LIN {X 0,Y 305.687,Z 241.405,A -85,B 0,C 180,E1 -15834.723,E2 -15834.723} C_VEL
LIN {X 0,Y 305.955,Z 241.369,A -85,B 0,C 180,E1 -15838.684,E2 -15838.684} C_VEL
LIN {X 0,Y 305.953,Z 241.364,A -85,B 0,C 180,E1 -15841.316,E2 -15841.316} C_VEL
LIN {X 0,Y 305.687,Z 241.402,A -85,B 0,C 180,E1 -15845.276,E2 -15845.276} C_VEL
LIN {X 0,Y 305.811,Z 241.392,A -85,B 0,C 180,E1 -15847.926,E2 -15847.926} C_VEL
LIN {X 0,Y 305.601,Z 241.415,A -85,B 0,C 180,E1 -15851.945,E2 -15851.945} C_VEL
LIN {X 0,Y 305.635,Z 241.408,A -85,B 0,C 180,E1 -15855.035,E2 -15855.035} C_VEL
LIN {X 0,Y 305.575,Z 241.418,A -85,B 0,C 180,E1 -15859.445,E2 -15859.445} C_VEL
LIN {X 0,Y 305.489,Z 241.428,A -85,B 0,C 180,E1 -15863.042,E2 -15863.042} C_VEL
LIN {X 0,Y 305.545,Z 241.427,A -85,B 0,C 180,E1 -15866.227,E2 -15866.227} C_VEL
LIN {X 0,Y 305.493,Z 241.428,A -85,B 0,C 180,E1 -15869.05,E2 -15869.05} C_VEL
LIN {X 0,Y 305.442,Z 241.437,A -85,B 0,C 180,E1 -15871.952,E2 -15871.952} C_VEL
LIN {X 0,Y 305.46,Z 241.433,A -85,B 0,C 180,E1 -15875.114,E2 -15875.114} C_VEL
LIN {X 0,Y 305.448,Z 241.439,A -85,B 0,C 180,E1 -15878.529,E2 -15878.529} C_VEL
LIN {X 0,Y 305.453,Z 241.434,A -85,B 0,C 180,E1 -15882.586,E2 -15882.586} C_VEL
LIN {X 0,Y 305.472,Z 241.432,A -85,B 0,C 180,E1 -15887.411,E2 -15887.411} C_VEL
LIN {X 0,Y 305.495,Z 241.428,A -85,B 0,C 180,E1 -15891.601,E2 -15891.601} C_VEL
LIN {X 0,Y 305.462,Z 241.439,A -85,B 0,C 180,E1 -15894.887,E2 -15894.887} C_VEL
LIN {X 0,Y 305.506,Z 241.55,A -85,B 0,C 180,E1 -15897.52,E2 -15897.52} C_VEL
LIN {X 0,Y 307.816,Z 252.02,A -85,B 0,C 180,E1 -15900.845,E2 -15900.845} C_VEL
LIN {X 0,Y 309.592,Z 261.539,A -85,B 0,C 180,E1 -15903.726,E2 -15903.726} C_VEL
LIN {X 0,Y 309.871,Z 264.214,A -85,B 0,C 180,E1 -15904.504,E2 -15904.504} C_VEL
LIN {X 0,Y 315.45,Z 298.867,A -85,B 0,C 180,E1 -15905.809,E2 -15905.809} C_VEL
LIN {X 0,Y 316.306,Z 306.855,A -85,B 0,C 180,E1 -15906.07,E2 -15906.07} C_VEL
LIN {X 0,Y 314.598,Z 373.309,A -85,B 0,C 180,E1 -15907.645,E2 -15907.645} C_VEL
LIN {X 0,Y 313.755,Z 386.795,A -85,B 0,C 180,E1 -15908.223,E2 -15908.223} C_VEL
LIN {X 0,Y 312.61,Z 399.148,A -85,B 0,C 180,E1 -15909.004,E2 -15909.004} C_VEL
LIN {X 0,Y 311.362,Z 411.031,A -85,B 0,C 180,E1 -15910.038,E2 -15910.038} C_VEL
LIN {X 0,Y 309.959,Z 422.47,A -85,B 0,C 180,E1 -15911.321,E2 -15911.321} C_VEL
LIN {X 0,Y 308.58,Z 432.784,A -85,B 0,C 180,E1 -15912.778,E2 -15912.778} C_VEL
LIN {X 0,Y 307.385,Z 442.048,A -85,B 0,C 180,E1 -15914.416,E2 -15914.416} C_VEL
LIN {X 0,Y 306.04,Z 451.048,A -85,B 0,C 180,E1 -15916.386,E2 -15916.386} C_VEL
LIN {X 0,Y 304.97,Z 458.282,A -85,B 0,C 180,E1 -15918.367,E2 -15918.367} C_VEL
LIN {X 0,Y 304.41,Z 463.162,A -85,B 0,C 180,E1 -15920.029,E2 -15920.029} C_VEL
LIN {X 0,Y 303.949,Z 467.893,A -85,B 0,C 180,E1 -15922.026,E2 -15922.026} C_VEL
LIN {X 0,Y 303.625,Z 472.136,A -85,B 0,C 180,E1 -15924.456,E2 -15924.456} C_VEL
LIN {X 0,Y 303.63,Z 474.065,A -85,B 0,C 180,E1 -15926.018,E2 -15926.018} C_VEL
LIN {X 0,Y 303.607,Z 475.267,A -85,B 0,C 180,E1 -15927.347,E2 -15927.347} C_VEL
LIN {X 0,Y 303.574,Z 476.018,A -85,B 0,C 180,E1 -15928.674,E2 -15928.674} C_VEL
LIN {X 0,Y 303.603,Z 476.368,A -85,B 0,C 180,E1 -15930,E2 -15930} C_VEL
LIN {X 0,Y 303.602,Z 475.896,A -85,B 0,C 180,E1 -15932.654,E2 -15932.654} C_VEL
LIN {X 0,Y 303.592,Z 475.028,A -85,B 0,C 180,E1 -15933.982,E2 -15933.982} C_VEL
LIN {X 0,Y 303.739,Z 472.071,A -85,B 0,C 180,E1 -15936.644,E2 -15936.644} C_VEL
LIN {X 0,Y 304.142,Z 468.709,A -85,B 0,C 180,E1 -15938.639,E2 -15938.639} C_VEL
LIN {X 0,Y 304.728,Z 464.278,A -85,B 0,C 180,E1 -15940.632,E2 -15940.632} C_VEL
LIN {X 0,Y 305.609,Z 458.66,A -85,B 0,C 180,E1 -15942.619,E2 -15942.619} C_VEL
LIN {X 0,Y 306.952,Z 451.662,A -85,B 0,C 180,E1 -15944.588,E2 -15944.588} C_VEL
LIN {X 0,Y 308.292,Z 443.612,A -85,B 0,C 180,E1 -15946.41,E2 -15946.41} C_VEL
LIN {X 0,Y 309.891,Z 433.972,A -85,B 0,C 180,E1 -15948.17,E2 -15948.17} C_VEL
LIN {X 0,Y 311.519,Z 424.167,A -85,B 0,C 180,E1 -15949.608,E2 -15949.608} C_VEL
LIN {X 0,Y 313.136,Z 413.41,A -85,B 0,C 180,E1 -15950.873,E2 -15950.873} C_VEL
LIN {X 0,Y 314.748,Z 401.372,A -85,B 0,C 180,E1 -15951.963,E2 -15951.963} C_VEL
LIN {X 0,Y 316.079,Z 388.872,A -85,B 0,C 180,E1 -15952.813,E2 -15952.813} C_VEL
LIN {X 0,Y 317.128,Z 375.767,A -85,B 0,C 180,E1 -15953.423,E2 -15953.423} C_VEL
LIN {X 0,Y 317.823,Z 359.088,A -85,B 0,C 180,E1 -15953.878,E2 -15953.878} C_VEL
LIN {X 0,Y 319.113,Z 304.9,A -85,B 0,C 180,E1 -15955.164,E2 -15955.164} C_VEL
LIN {X 0,Y 315.677,Z 283.465,A -85,B 0,C 180,E1 -15956.063,E2 -15956.063} C_VEL
LIN {X 0,Y 312.582,Z 268.833,A -85,B 0,C 180,E1 -15956.769,E2 -15956.769} C_VEL
LIN {X 0,Y 310.331,Z 263.131,A -85,B 0,C 180,E1 -15957.165,E2 -15957.165} C_VEL
LIN {X 0,Y 308.466,Z 253.823,A -85,B 0,C 180,E1 -15960.082,E2 -15960.082} C_VEL
LIN {X 0,Y 306.055,Z 243.759,A -85,B 0,C 180,E1 -15963.444,E2 -15963.444} C_VEL
LIN {X 0,Y 305.478,Z 241.436,A -85,B 0,C 180,E1 -15964.32,E2 -15964.32} C_VEL
LIN {X 0,Y 305.476,Z 241.432,A -85,B 0,C 180,E1 -15968.402,E2 -15968.402} C_VEL
LIN {X 0,Y 305.455,Z 241.433,A -85,B 0,C 180,E1 -15972.586,E2 -15972.586} C_VEL
LIN {X 0,Y 305.426,Z 241.441,A -85,B 0,C 180,E1 -15976.345,E2 -15976.345} C_VEL
LIN {X 0,Y 305.458,Z 241.436,A -85,B 0,C 180,E1 -15979.892,E2 -15979.892} C_VEL
LIN {X 0,Y 305.481,Z 241.431,A -85,B 0,C 180,E1 -15983.631,E2 -15983.631} C_VEL
LIN {X 0,Y 305.465,Z 241.433,A -85,B 0,C 180,E1 -15986.483,E2 -15986.483} C_VEL
LIN {X 0,Y 305.458,Z 241.432,A -85,B 0,C 180,E1 -15989.59,E2 -15989.59} C_VEL
LIN {X 0,Y 305.518,Z 241.42,A -85,B 0,C 180,E1 -15992.608,E2 -15992.608} C_VEL
LIN {X 0,Y 305.508,Z 241.427,A -85,B 0,C 180,E1 -15995.539,E2 -15995.539} C_VEL
LIN {X 0,Y 305.519,Z 241.426,A -85,B 0,C 180,E1 -15999.815,E2 -15999.815} C_VEL
LIN {X 0,Y 305.574,Z 241.416,A -85,B 0,C 180,E1 -16002.603,E2 -16002.603} C_VEL
LIN {X 0,Y 305.649,Z 241.401,A -85,B 0,C 180,E1 -16005.349,E2 -16005.349} C_VEL
LIN {X 0,Y 305.638,Z 241.407,A -85,B 0,C 180,E1 -16009.4,E2 -16009.4} C_VEL
LIN {X 0,Y 305.808,Z 241.389,A -85,B 0,C 180,E1 -16012.074,E2 -16012.074} C_VEL
LIN {X 0,Y 305.686,Z 241.399,A -85,B 0,C 180,E1 -16014.724,E2 -16014.724} C_VEL
LIN {X 0,Y 305.955,Z 241.369,A -85,B 0,C 180,E1 -16018.684,E2 -16018.684} C_VEL
LIN {X 0,Y 305.957,Z 241.374,A -85,B 0,C 180,E1 -16021.316,E2 -16021.316} C_VEL
LIN {X 0,Y 305.851,Z 241.387,A -85,B 0,C 180,E1 -16026.598,E2 -16026.598} C_VEL
LIN {X 0,Y 305.736,Z 241.401,A -85,B 0,C 180,E1 -16029.26,E2 -16029.26} C_VEL
LIN {X 0,Y 305.589,Z 241.42,A -85,B 0,C 180,E1 -16033.296,E2 -16033.296} C_VEL
LIN {X 0,Y 305.594,Z 241.415,A -85,B 0,C 180,E1 -16036.02,E2 -16036.02} C_VEL
LIN {X 0,Y 305.576,Z 241.421,A -85,B 0,C 180,E1 -16039.444,E2 -16039.444} C_VEL
LIN {X 0,Y 305.486,Z 241.432,A -85,B 0,C 180,E1 -16043.04,E2 -16043.04} C_VEL
LIN {X 0,Y 305.478,Z 241.432,A -85,B 0,C 180,E1 -16046.201,E2 -16046.201} C_VEL
LIN {X 0,Y 305.463,Z 241.425,A -85,B 0,C 180,E1 -16049.039,E2 -16049.039} C_VEL
LIN {X 0,Y 305.437,Z 241.433,A -85,B 0,C 180,E1 -16051.953,E2 -16051.953} C_VEL
LIN {X 0,Y 305.509,Z 241.449,A -85,B 0,C 180,E1 -16054.963,E2 -16054.963} C_VEL
LIN {X 0,Y 307.325,Z 248.984,A -85,B 0,C 180,E1 -16057.56,E2 -16057.56} C_VEL
LIN {X 0,Y 314.914,Z 265.656,A -85,B 0,C 180,E1 -16058.826,E2 -16058.826} C_VEL
LIN {X 0,Y 318.632,Z 275.459,A -85,B 0,C 180,E1 -16059.458,E2 -16059.458} C_VEL
LIN {X 0,Y 319.852,Z 282.666,A -85,B 0,C 180,E1 -16059.766,E2 -16059.766} C_VEL
LIN {X 0,Y 317.555,Z 356.862,A -85,B 0,C 180,E1 -16061.521,E2 -16061.521} C_VEL
LIN {X 0,Y 316.73,Z 370.282,A -85,B 0,C 180,E1 -16062.098,E2 -16062.098} C_VEL
LIN {X 0,Y 315.633,Z 382.988,A -85,B 0,C 180,E1 -16062.909,E2 -16062.909} C_VEL
LIN {X 0,Y 314.192,Z 395.492,A -85,B 0,C 180,E1 -16064.007,E2 -16064.007} C_VEL
LIN {X 0,Y 312.768,Z 405.819,A -85,B 0,C 180,E1 -16065.17,E2 -16065.17} C_VEL
LIN {X 0,Y 311.245,Z 415.778,A -85,B 0,C 180,E1 -16066.566,E2 -16066.566} C_VEL
LIN {X 0,Y 309.825,Z 423.975,A -85,B 0,C 180,E1 -16067.969,E2 -16067.969} C_VEL
LIN {X 0,Y 308.179,Z 433.065,A -85,B 0,C 180,E1 -16069.891,E2 -16069.891} C_VEL
LIN {X 0,Y 306.879,Z 440.278,A -85,B 0,C 180,E1 -16071.805,E2 -16071.805} C_VEL
LIN {X 0,Y 305.889,Z 445.559,A -85,B 0,C 180,E1 -16073.528,E2 -16073.528} C_VEL
LIN {X 0,Y 304.994,Z 450.479,A -85,B 0,C 180,E1 -16075.539,E2 -16075.539} C_VEL
LIN {X 0,Y 304.303,Z 454.817,A -85,B 0,C 180,E1 -16077.914,E2 -16077.914} C_VEL
LIN {X 0,Y 303.94,Z 456.818,A -85,B 0,C 180,E1 -16079.422,E2 -16079.422} C_VEL
LIN {X 0,Y 303.555,Z 458.759,A -85,B 0,C 180,E1 -16081.618,E2 -16081.618} C_VEL
LIN {X 0,Y 303.342,Z 459.607,A -85,B 0,C 180,E1 -16083.883,E2 -16083.883} C_VEL
LIN {X 0,Y 303.31,Z 459.554,A -85,B 0,C 180,E1 -16085.35,E2 -16085.35} C_VEL
LIN {X 0,Y 303.408,Z 458.277,A -85,B 0,C 180,E1 -16087.903,E2 -16087.903} C_VEL
LIN {X 0,Y 303.822,Z 455.551,A -85,B 0,C 180,E1 -16090.402,E2 -16090.402} C_VEL
LIN {X 0,Y 304.263,Z 452.031,A -85,B 0,C 180,E1 -16092.526,E2 -16092.526} C_VEL
LIN {X 0,Y 304.826,Z 447.343,A -85,B 0,C 180,E1 -16094.625,E2 -16094.625} C_VEL
LIN {X 0,Y 305.708,Z 441.312,A -85,B 0,C 180,E1 -16096.709,E2 -16096.709} C_VEL
LIN {X 0,Y 306.77,Z 433.714,A -85,B 0,C 180,E1 -16098.771,E2 -16098.771} C_VEL
LIN {X 0,Y 307.949,Z 425.894,A -85,B 0,C 180,E1 -16100.482,E2 -16100.482} C_VEL
LIN {X 0,Y 309.248,Z 416.482,A -85,B 0,C 180,E1 -16102.163,E2 -16102.163} C_VEL
LIN {X 0,Y 310.677,Z 405.452,A -85,B 0,C 180,E1 -16103.726,E2 -16103.726} C_VEL
LIN {X 0,Y 312.054,Z 394.084,A -85,B 0,C 180,E1 -16104.993,E2 -16104.993} C_VEL
LIN {X 0,Y 313.249,Z 381.694,A -85,B 0,C 180,E1 -16106.06,E2 -16106.06} C_VEL
LIN {X 0,Y 314.143,Z 368.704,A -85,B 0,C 180,E1 -16106.874,E2 -16106.874} C_VEL
LIN {X 0,Y 314.773,Z 356.239,A -85,B 0,C 180,E1 -16107.4,E2 -16107.4} C_VEL
LIN {X 0,Y 316.733,Z 280.316,A -85,B 0,C 180,E1 -16109.187,E2 -16109.187} C_VEL
LIN {X 0,Y 314.043,Z 267.159,A -85,B 0,C 180,E1 -16109.718,E2 -16109.718} C_VEL
LIN {X 0,Y 307.327,Z 248.529,A -85,B 0,C 180,E1 -16110.737,E2 -16110.737} C_VEL
LIN {X 0,Y 305.729,Z 241.405,A -85,B 0,C 180,E1 -16113.212,E2 -16113.212} C_VEL
LIN {X 0,Y 305.789,Z 241.395,A -85,B 0,C 180,E1 -16116.599,E2 -16116.599} C_VEL
LIN {X 0,Y 305.696,Z 241.406,A -85,B 0,C 180,E1 -16119.261,E2 -16119.261} C_VEL
LIN {X 0,Y 305.591,Z 241.419,A -85,B 0,C 180,E1 -16123.296,E2 -16123.296} C_VEL
LIN {X 0,Y 305.596,Z 241.421,A -85,B 0,C 180,E1 -16126.02,E2 -16126.02} C_VEL
LIN {X 0,Y 305.577,Z 241.422,A -85,B 0,C 180,E1 -16129.444,E2 -16129.444} C_VEL
LIN {X 0,Y 305.487,Z 241.427,A -85,B 0,C 180,E1 -16133.039,E2 -16133.039} C_VEL
LIN {X 0,Y 305.476,Z 241.433,A -85,B 0,C 180,E1 -16136.199,E2 -16136.199} C_VEL
LIN {X 0,Y 305.459,Z 241.43,A -85,B 0,C 180,E1 -16139.037,E2 -16139.037} C_VEL
LIN {X 0,Y 305.437,Z 241.441,A -85,B 0,C 180,E1 -16141.952,E2 -16141.952} C_VEL
LIN {X 0,Y 305.462,Z 241.43,A -85,B 0,C 180,E1 -16145.113,E2 -16145.113} C_VEL
LIN {X 0,Y 305.466,Z 241.433,A -85,B 0,C 180,E1 -16148.532,E2 -16148.532} C_VEL
LIN {X 0,Y 305.454,Z 241.431,A -85,B 0,C 180,E1 -16152.585,E2 -16152.585} C_VEL
LIN {X 0,Y 305.425,Z 241.438,A -85,B 0,C 180,E1 -16156.344,E2 -16156.344} C_VEL
LIN {X 0,Y 305.457,Z 241.438,A -85,B 0,C 180,E1 -16159.892,E2 -16159.892} C_VEL
LIN {X 0,Y 305.458,Z 241.432,A -85,B 0,C 180,E1 -16161.37,E2 -16161.37} C_VEL
LIN {X 0,Y 304.851,Z 241.512,A -85,B 0,C 180,E1 -16162.47,E2 -16162.47} C_VEL
LIN {X 0,Y 302.014,Z 241.864,A -85,B 0,C 180,E1 -16164.26,E2 -16164.26} C_VEL
LIN {X 0,Y 299.559,Z 242.166,A -85,B 0,C 180,E1 -16165.713,E2 -16165.713} C_VEL
LIN {X 0,Y 298.488,Z 242.299,A -85,B 0,C 180,E1 -16166.838,E2 -16166.838} C_VEL
LIN {X 0,Y 298.393,Z 242.311,A -85,B 0,C 180,E1 -16167.22,E2 -16167.22} C_VEL
LIN {X 0,Y 298.457,Z 242.309,A -85,B 0,C 180,E1 -16171.903,E2 -16171.903} C_VEL
LIN {X 0,Y 298.484,Z 242.294,A -85,B 0,C 180,E1 -16174.924,E2 -16174.924} C_VEL
LIN {X 0,Y 298.448,Z 242.303,A -85,B 0,C 180,E1 -16179.315,E2 -16179.315} C_VEL
LIN {X 0,Y 298.536,Z 242.3,A -85,B 0,C 180,E1 -16182.179,E2 -16182.179} C_VEL
LIN {X 0,Y 298.591,Z 242.286,A -85,B 0,C 180,E1 -16184.994,E2 -16184.994} C_VEL
LIN {X 0,Y 298.591,Z 242.277,A -85,B 0,C 180,E1 -16189.146,E2 -16189.146} C_VEL
LIN {X 0,Y 298.756,Z 242.266,A -85,B 0,C 180,E1 -16191.886,E2 -16191.886} C_VEL
LIN {X 0,Y 298.658,Z 242.282,A -85,B 0,C 180,E1 -16194.599,E2 -16194.599} C_VEL
LIN {X 0,Y 298.921,Z 242.245,A -85,B 0,C 180,E1 -16198.653,E2 -16198.653} C_VEL
LIN {X 0,Y 298.92,Z 242.239,A -85,B 0,C 180,E1 -16201.347,E2 -16201.347} C_VEL
LIN {X 0,Y 298.796,Z 242.264,A -85,B 0,C 180,E1 -16206.754,E2 -16206.754} C_VEL
LIN {X 0,Y 298.678,Z 242.277,A -85,B 0,C 180,E1 -16209.48,E2 -16209.48} C_VEL
LIN {X 0,Y 298.549,Z 242.286,A -85,B 0,C 180,E1 -16213.615,E2 -16213.615} C_VEL
LIN {X 0,Y 298.546,Z 242.297,A -85,B 0,C 180,E1 -16216.409,E2 -16216.409} C_VEL
LIN {X 0,Y 298.51,Z 242.299,A -85,B 0,C 180,E1 -16219.655,E2 -16219.655} C_VEL
LIN {X 0,Y 298.456,Z 242.304,A -85,B 0,C 180,E1 -16223.598,E2 -16223.598} C_VEL
LIN {X 0,Y 298.487,Z 242.303,A -85,B 0,C 180,E1 -16226.575,E2 -16226.575} C_VEL
LIN {X 0,Y 298.419,Z 242.309,A -85,B 0,C 180,E1 -16229.641,E2 -16229.641} C_VEL
LIN {X 0,Y 298.394,Z 242.313,A -85,B 0,C 180,E1 -16232.8,E2 -16232.8} C_VEL
LIN {X 0,Y 298.444,Z 242.308,A -85,B 0,C 180,E1 -16236.808,E2 -16236.808} C_VEL
LIN {X 0,Y 298.385,Z 242.313,A -85,B 0,C 180,E1 -16241.088,E2 -16241.088} C_VEL
LIN {X 0,Y 298.397,Z 242.311,A -85,B 0,C 180,E1 -16243.104,E2 -16243.104} C_VEL
LIN {X 0,Y 298.402,Z 242.314,A -85,B 0,C 180,E1 -16246.921,E2 -16246.921} C_VEL
LIN {X 0,Y 298.414,Z 242.31,A -85,B 0,C 180,E1 -16251.004,E2 -16251.004} C_VEL
LIN {X 0,Y 298.432,Z 242.312,A -85,B 0,C 180,E1 -16253.933,E2 -16253.933} C_VEL
LIN {X 0,Y 298.47,Z 242.508,A -85,B 0,C 180,E1 -16257.109,E2 -16257.109} C_VEL
LIN {X 0,Y 301.138,Z 254.596,A -85,B 0,C 180,E1 -16261.036,E2 -16261.036} C_VEL
LIN {X 0,Y 302.819,Z 263.96,A -85,B 0,C 180,E1 -16263.92,E2 -16263.92} C_VEL
LIN {X 0,Y 304.316,Z 270.953,A -85,B 0,C 180,E1 -16264.248,E2 -16264.248} C_VEL
LIN {X 0,Y 309.005,Z 300.828,A -85,B 0,C 180,E1 -16265.389,E2 -16265.389} C_VEL
LIN {X 0,Y 309.698,Z 307.298,A -85,B 0,C 180,E1 -16265.606,E2 -16265.606} C_VEL
LIN {X 0,Y 307.961,Z 372.416,A -85,B 0,C 180,E1 -16267.173,E2 -16267.173} C_VEL
LIN {X 0,Y 307.143,Z 385.493,A -85,B 0,C 180,E1 -16267.73,E2 -16267.73} C_VEL
LIN {X 0,Y 305.974,Z 398.155,A -85,B 0,C 180,E1 -16268.527,E2 -16268.527} C_VEL
LIN {X 0,Y 304.687,Z 410.258,A -85,B 0,C 180,E1 -16269.582,E2 -16269.582} C_VEL
LIN {X 0,Y 303.202,Z 421.801,A -85,B 0,C 180,E1 -16270.889,E2 -16270.889} C_VEL
LIN {X 0,Y 301.734,Z 432.211,A -85,B 0,C 180,E1 -16272.375,E2 -16272.375} C_VEL
LIN {X 0,Y 300.518,Z 441.564,A -85,B 0,C 180,E1 -16274.051,E2 -16274.051} C_VEL
LIN {X 0,Y 299.121,Z 450.617,A -85,B 0,C 180,E1 -16276.065,E2 -16276.065} C_VEL
LIN {X 0,Y 297.977,Z 457.899,A -85,B 0,C 180,E1 -16278.09,E2 -16278.09} C_VEL
LIN {X 0,Y 297.395,Z 462.814,A -85,B 0,C 180,E1 -16279.791,E2 -16279.791} C_VEL
LIN {X 0,Y 296.889,Z 467.578,A -85,B 0,C 180,E1 -16281.835,E2 -16281.835} C_VEL
LIN {X 0,Y 296.687,Z 470.134,A -85,B 0,C 180,E1 -16283.198,E2 -16283.198} C_VEL
LIN {X 0,Y 296.552,Z 472.182,A -85,B 0,C 180,E1 -16284.561,E2 -16284.561} C_VEL
LIN {X 0,Y 296.528,Z 473.81,A -85,B 0,C 180,E1 -16285.923,E2 -16285.923} C_VEL
LIN {X 0,Y 296.533,Z 475.028,A -85,B 0,C 180,E1 -16287.283,E2 -16287.283} C_VEL
LIN {X 0,Y 296.493,Z 475.802,A -85,B 0,C 180,E1 -16288.642,E2 -16288.642} C_VEL
LIN {X 0,Y 296.518,Z 476.165,A -85,B 0,C 180,E1 -16290,E2 -16290} C_VEL
LIN {X 0,Y 296.526,Z 475.72,A -85,B 0,C 180,E1 -16292.717,E2 -16292.717} C_VEL
LIN {X 0,Y 296.492,Z 474.876,A -85,B 0,C 180,E1 -16294.078,E2 -16294.078} C_VEL
LIN {X 0,Y 296.687,Z 471.947,A -85,B 0,C 180,E1 -16296.802,E2 -16296.802} C_VEL
LIN {X 0,Y 297.085,Z 468.613,A -85,B 0,C 180,E1 -16298.845,E2 -16298.845} C_VEL
LIN {X 0,Y 297.73,Z 464.212,A -85,B 0,C 180,E1 -16300.885,E2 -16300.885} C_VEL
LIN {X 0,Y 298.667,Z 458.625,A -85,B 0,C 180,E1 -16302.918,E2 -16302.918} C_VEL
LIN {X 0,Y 300.086,Z 451.669,A -85,B 0,C 180,E1 -16304.929,E2 -16304.929} C_VEL
LIN {X 0,Y 301.424,Z 443.978,A -85,B 0,C 180,E1 -16306.73,E2 -16306.73} C_VEL
LIN {X 0,Y 303.133,Z 434.09,A -85,B 0,C 180,E1 -16308.59,E2 -16308.59} C_VEL
LIN {X 0,Y 304.841,Z 424.365,A -85,B 0,C 180,E1 -16310.056,E2 -16310.056} C_VEL
LIN {X 0,Y 306.544,Z 413.741,A -85,B 0,C 180,E1 -16311.344,E2 -16311.344} C_VEL
LIN {X 0,Y 308.204,Z 401.89,A -85,B 0,C 180,E1 -16312.455,E2 -16312.455} C_VEL
LIN {X 0,Y 309.597,Z 389.631,A -85,B 0,C 180,E1 -16313.318,E2 -16313.318} C_VEL
LIN {X 0,Y 310.635,Z 377.158,A -85,B 0,C 180,E1 -16313.943,E2 -16313.943} C_VEL
LIN {X 0,Y 311.325,Z 363.499,A -85,B 0,C 180,E1 -16314.356,E2 -16314.356} C_VEL
LIN {X 0,Y 312.846,Z 305.915,A -85,B 0,C 180,E1 -16315.744,E2 -16315.744} C_VEL
LIN {X 0,Y 309.358,Z 284.053,A -85,B 0,C 180,E1 -16316.689,E2 -16316.689} C_VEL
LIN {X 0,Y 306.78,Z 271.703,A -85,B 0,C 180,E1 -16317.306,E2 -16317.306} C_VEL
LIN {X 0,Y 303.184,Z 262.833,A -85,B 0,C 180,E1 -16317.975,E2 -16317.975} C_VEL
LIN {X 0,Y 300.996,Z 252.678,A -85,B 0,C 180,E1 -16321.3,E2 -16321.3} C_VEL
LIN {X 0,Y 298.437,Z 242.314,A -85,B 0,C 180,E1 -16324.978,E2 -16324.978} C_VEL
LIN {X 0,Y 298.414,Z 242.311,A -85,B 0,C 180,E1 -16327.758,E2 -16327.758} C_VEL
LIN {X 0,Y 298.386,Z 242.32,A -85,B 0,C 180,E1 -16331.261,E2 -16331.261} C_VEL
LIN {X 0,Y 298.354,Z 242.319,A -85,B 0,C 180,E1 -16335.035,E2 -16335.035} C_VEL
LIN {X 0,Y 298.384,Z 242.313,A -85,B 0,C 180,E1 -16338.738,E2 -16338.738} C_VEL
LIN {X 0,Y 298.414,Z 242.311,A -85,B 0,C 180,E1 -16342.242,E2 -16342.242} C_VEL
LIN {X 0,Y 298.408,Z 242.309,A -85,B 0,C 180,E1 -16345.581,E2 -16345.581} C_VEL
LIN {X 0,Y 298.391,Z 242.307,A -85,B 0,C 180,E1 -16348.791,E2 -16348.791} C_VEL
LIN {X 0,Y 298.459,Z 242.301,A -85,B 0,C 180,E1 -16351.904,E2 -16351.904} C_VEL
LIN {X 0,Y 298.485,Z 242.306,A -85,B 0,C 180,E1 -16354.924,E2 -16354.924} C_VEL
LIN {X 0,Y 298.45,Z 242.309,A -85,B 0,C 180,E1 -16359.315,E2 -16359.315} C_VEL
LIN {X 0,Y 298.538,Z 242.29,A -85,B 0,C 180,E1 -16362.179,E2 -16362.179} C_VEL
LIN {X 0,Y 298.593,Z 242.283,A -85,B 0,C 180,E1 -16364.995,E2 -16364.995} C_VEL
LIN {X 0,Y 298.593,Z 242.286,A -85,B 0,C 180,E1 -16369.147,E2 -16369.147} C_VEL
LIN {X 0,Y 298.755,Z 242.267,A -85,B 0,C 180,E1 -16371.886,E2 -16371.886} C_VEL
LIN {X 0,Y 298.657,Z 242.275,A -85,B 0,C 180,E1 -16374.599,E2 -16374.599} C_VEL
LIN {X 0,Y 298.922,Z 242.245,A -85,B 0,C 180,E1 -16378.653,E2 -16378.653} C_VEL
LIN {X 0,Y 298.923,Z 242.25,A -85,B 0,C 180,E1 -16381.347,E2 -16381.347} C_VEL
LIN {X 0,Y 298.797,Z 242.264,A -85,B 0,C 180,E1 -16386.754,E2 -16386.754} C_VEL
LIN {X 0,Y 298.681,Z 242.279,A -85,B 0,C 180,E1 -16389.481,E2 -16389.481} C_VEL
LIN {X 0,Y 298.552,Z 242.296,A -85,B 0,C 180,E1 -16393.616,E2 -16393.616} C_VEL
LIN {X 0,Y 298.549,Z 242.295,A -85,B 0,C 180,E1 -16396.409,E2 -16396.409} C_VEL
LIN {X 0,Y 298.51,Z 242.301,A -85,B 0,C 180,E1 -16399.654,E2 -16399.654} C_VEL
LIN {X 0,Y 298.424,Z 242.309,A -85,B 0,C 180,E1 -16403.601,E2 -16403.601} C_VEL
LIN {X 0,Y 298.417,Z 242.313,A -85,B 0,C 180,E1 -16406.582,E2 -16406.582} C_VEL
LIN {X 0,Y 298.4,Z 242.307,A -85,B 0,C 180,E1 -16409.643,E2 -16409.643} C_VEL
LIN {X 0,Y 298.429,Z 242.316,A -85,B 0,C 180,E1 -16414.008,E2 -16414.008} C_VEL
LIN {X 0,Y 298.459,Z 242.457,A -85,B 0,C 180,E1 -16414.31,E2 -16414.31} C_VEL
LIN {X 0,Y 300.19,Z 249.338,A -85,B 0,C 180,E1 -16416.751,E2 -16416.751} C_VEL
LIN {X 0,Y 308.088,Z 266.098,A -85,B 0,C 180,E1 -16418.123,E2 -16418.123} C_VEL
LIN {X 0,Y 312.595,Z 277.605,A -85,B 0,C 180,E1 -16418.911,E2 -16418.911} C_VEL
LIN {X 0,Y 313.595,Z 283.802,A -85,B 0,C 180,E1 -16419.179,E2 -16419.179} C_VEL
LIN {X 0,Y 311.226,Z 357.088,A -85,B 0,C 180,E1 -16420.947,E2 -16420.947} C_VEL
LIN {X 0,Y 310.36,Z 370.355,A -85,B 0,C 180,E1 -16421.524,E2 -16421.524} C_VEL
LIN {X 0,Y 309.171,Z 383.4,A -85,B 0,C 180,E1 -16422.372,E2 -16422.372} C_VEL
LIN {X 0,Y 307.664,Z 396.004,A -85,B 0,C 180,E1 -16423.509,E2 -16423.509} C_VEL
LIN {X 0,Y 306.09,Z 406.928,A -85,B 0,C 180,E1 -16424.779,E2 -16424.779} C_VEL
LIN {X 0,Y 304.527,Z 416.586,A -85,B 0,C 180,E1 -16426.183,E2 -16426.183} C_VEL
LIN {X 0,Y 302.927,Z 425.191,A -85,B 0,C 180,E1 -16427.716,E2 -16427.716} C_VEL
LIN {X 0,Y 301.307,Z 433.724,A -85,B 0,C 180,E1 -16429.599,E2 -16429.599} C_VEL
LIN {X 0,Y 299.902,Z 441.042,A -85,B 0,C 180,E1 -16431.61,E2 -16431.61} C_VEL
LIN {X 0,Y 298.563,Z 447.718,A -85,B 0,C 180,E1 -16433.95,E2 -16433.95} C_VEL
LIN {X 0,Y 297.627,Z 452.853,A -85,B 0,C 180,E1 -16436.373,E2 -16436.373} C_VEL
LIN {X 0,Y 297.031,Z 456.301,A -85,B 0,C 180,E1 -16438.632,E2 -16438.632} C_VEL
LIN {X 0,Y 296.523,Z 458.842,A -85,B 0,C 180,E1 -16441.277,E2 -16441.277} C_VEL
LIN {X 0,Y 296.294,Z 459.721,A -85,B 0,C 180,E1 -16443.213,E2 -16443.213} C_VEL
LIN {X 0,Y 296.225,Z 459.828,A -85,B 0,C 180,E1 -16444.719,E2 -16444.719} C_VEL
LIN {X 0,Y 296.214,Z 459.465,A -85,B 0,C 180,E1 -16446.213,E2 -16446.213} C_VEL
LIN {X 0,Y 296.3,Z 458.651,A -85,B 0,C 180,E1 -16447.697,E2 -16447.697} C_VEL
LIN {X 0,Y 296.463,Z 457.318,A -85,B 0,C 180,E1 -16449.17,E2 -16449.17} C_VEL
LIN {X 0,Y 296.923,Z 454.66,A -85,B 0,C 180,E1 -16451.224,E2 -16451.224} C_VEL
LIN {X 0,Y 297.393,Z 450.451,A -85,B 0,C 180,E1 -16453.526,E2 -16453.526} C_VEL
LIN {X 0,Y 298.155,Z 444.836,A -85,B 0,C 180,E1 -16455.815,E2 -16455.815} C_VEL
LIN {X 0,Y 299.104,Z 438.617,A -85,B 0,C 180,E1 -16457.791,E2 -16457.791} C_VEL
LIN {X 0,Y 300.287,Z 431.048,A -85,B 0,C 180,E1 -16459.716,E2 -16459.716} C_VEL
LIN {X 0,Y 301.684,Z 421.701,A -85,B 0,C 180,E1 -16461.628,E2 -16461.628} C_VEL
LIN {X 0,Y 302.977,Z 412.361,A -85,B 0,C 180,E1 -16463.172,E2 -16463.172} C_VEL
LIN {X 0,Y 304.388,Z 402.197,A -85,B 0,C 180,E1 -16464.523,E2 -16464.523} C_VEL
LIN {X 0,Y 305.681,Z 390.91,A -85,B 0,C 180,E1 -16465.715,E2 -16465.715} C_VEL
LIN {X 0,Y 306.762,Z 378.631,A -85,B 0,C 180,E1 -16466.716,E2 -16466.716} C_VEL
LIN {X 0,Y 307.663,Z 365.902,A -85,B 0,C 180,E1 -16467.463,E2 -16467.463} C_VEL
LIN {X 0,Y 308.238,Z 352.723,A -85,B 0,C 180,E1 -16467.958,E2 -16467.958} C_VEL
LIN {X 0,Y 310.124,Z 281.133,A -85,B 0,C 180,E1 -16469.657,E2 -16469.657} C_VEL
LIN {X 0,Y 307.692,Z 269.305,A -85,B 0,C 180,E1 -16470.15,E2 -16470.15} C_VEL
LIN {X 0,Y 300.147,Z 248.795,A -85,B 0,C 180,E1 -16471.306,E2 -16471.306} C_VEL
LIN {X 0,Y 298.637,Z 242.29,A -85,B 0,C 180,E1 -16473.626,E2 -16473.626} C_VEL
LIN {X 0,Y 298.738,Z 242.274,A -85,B 0,C 180,E1 -16476.755,E2 -16476.755} C_VEL
LIN {X 0,Y 298.628,Z 242.288,A -85,B 0,C 180,E1 -16479.482,E2 -16479.482} C_VEL
LIN {X 0,Y 298.554,Z 242.298,A -85,B 0,C 180,E1 -16483.615,E2 -16483.615} C_VEL
LIN {X 0,Y 298.551,Z 242.297,A -85,B 0,C 180,E1 -16486.408,E2 -16486.408} C_VEL
LIN {X 0,Y 298.512,Z 242.304,A -85,B 0,C 180,E1 -16489.653,E2 -16489.653} C_VEL
LIN {X 0,Y 298.426,Z 242.309,A -85,B 0,C 180,E1 -16493.6,E2 -16493.6} C_VEL
LIN {X 0,Y 298.415,Z 242.31,A -85,B 0,C 180,E1 -16496.581,E2 -16496.581} C_VEL
LIN {X 0,Y 298.398,Z 242.313,A -85,B 0,C 180,E1 -16499.643,E2 -16499.643} C_VEL
LIN {X 0,Y 298.393,Z 242.313,A -85,B 0,C 180,E1 -16502.8,E2 -16502.8} C_VEL
LIN {X 0,Y 298.446,Z 242.304,A -85,B 0,C 180,E1 -16506.807,E2 -16506.807} C_VEL
LIN {X 0,Y 298.408,Z 242.313,A -85,B 0,C 180,E1 -16509.486,E2 -16509.486} C_VEL
LIN {X 0,Y 298.398,Z 242.309,A -85,B 0,C 180,E1 -16513.103,E2 -16513.103} C_VEL
LIN {X 0,Y 298.402,Z 242.311,A -85,B 0,C 180,E1 -16516.92,E2 -16516.92} C_VEL
LIN {X 0,Y 298.414,Z 242.309,A -85,B 0,C 180,E1 -16521.003,E2 -16521.003} C_VEL
LIN {X 0,Y 298.417,Z 242.307,A -85,B 0,C 180,E1 -16523.93,E2 -16523.93} C_VEL
LIN {X 0,Y 298.393,Z 242.311,A -85,B 0,C 180,E1 -16527.22,E2 -16527.22} C_VEL
LIN {X 0,Y 297.726,Z 242.398,A -85,B 0,C 180,E1 -16528.346,E2 -16528.346} C_VEL
LIN {X 0,Y 294.947,Z 242.748,A -85,B 0,C 180,E1 -16530.184,E2 -16530.184} C_VEL
LIN {X 0,Y 292.581,Z 243.041,A -85,B 0,C 180,E1 -16531.675,E2 -16531.675} C_VEL
LIN {X 0,Y 291.536,Z 243.166,A -85,B 0,C 180,E1 -16532.827,E2 -16532.827} C_VEL
LIN {X 0,Y 291.434,Z 243.176,A -85,B 0,C 180,E1 -16533.218,E2 -16533.218} C_VEL
LIN {X 0,Y 291.379,Z 243.178,A -85,B 0,C 180,E1 -16537.299,E2 -16537.299} C_VEL
LIN {X 0,Y 291.456,Z 243.18,A -85,B 0,C 180,E1 -16540.27,E2 -16540.27} C_VEL
LIN {X 0,Y 291.553,Z 243.164,A -85,B 0,C 180,E1 -16544.623,E2 -16544.623} C_VEL
LIN {X 0,Y 291.535,Z 243.155,A -85,B 0,C 180,E1 -16548.88,E2 -16548.88} C_VEL
LIN {X 0,Y 291.707,Z 243.142,A -85,B 0,C 180,E1 -16551.688,E2 -16551.688} C_VEL
LIN {X 0,Y 291.629,Z 243.158,A -85,B 0,C 180,E1 -16554.468,E2 -16554.468} C_VEL
LIN {X 0,Y 291.888,Z 243.121,A -85,B 0,C 180,E1 -16558.62,E2 -16558.62} C_VEL
LIN {X 0,Y 291.886,Z 243.115,A -85,B 0,C 180,E1 -16561.38,E2 -16561.38} C_VEL
LIN {X 0,Y 291.744,Z 243.141,A -85,B 0,C 180,E1 -16566.918,E2 -16566.918} C_VEL
LIN {X 0,Y 291.627,Z 243.157,A -85,B 0,C 180,E1 -16569.712,E2 -16569.712} C_VEL
LIN {X 0,Y 291.519,Z 243.163,A -85,B 0,C 180,E1 -16573.95,E2 -16573.95} C_VEL
LIN {X 0,Y 291.485,Z 243.174,A -85,B 0,C 180,E1 -16576.818,E2 -16576.818} C_VEL
LIN {X 0,Y 291.449,Z 243.18,A -85,B 0,C 180,E1 -16579.875,E2 -16579.875} C_VEL
LIN {X 0,Y 291.399,Z 243.187,A -85,B 0,C 180,E1 -16584.205,E2 -16584.205} C_VEL
LIN {X 0,Y 291.421,Z 243.181,A -85,B 0,C 180,E1 -16587.272,E2 -16587.272} C_VEL
LIN {X 0,Y 291.335,Z 243.197,A -85,B 0,C 180,E1 -16590.437,E2 -16590.437} C_VEL
LIN {X 0,Y 291.343,Z 243.19,A -85,B 0,C 180,E1 -16593.699,E2 -16593.699} C_VEL
LIN {X 0,Y 291.374,Z 243.187,A -85,B 0,C 180,E1 -16597.254,E2 -16597.254} C_VEL
LIN {X 0,Y 291.331,Z 243.194,A -85,B 0,C 180,E1 -16600.643,E2 -16600.643} C_VEL
LIN {X 0,Y 291.289,Z 243.201,A -85,B 0,C 180,E1 -16604.402,E2 -16604.402} C_VEL
LIN {X 0,Y 291.346,Z 243.195,A -85,B 0,C 180,E1 -16608.4,E2 -16608.4} C_VEL
LIN {X 0,Y 291.364,Z 243.188,A -85,B 0,C 180,E1 -16611.161,E2 -16611.161} C_VEL
LIN {X 0,Y 291.385,Z 243.191,A -85,B 0,C 180,E1 -16614.63,E2 -16614.63} C_VEL
LIN {X 0,Y 291.415,Z 243.328,A -85,B 0,C 180,E1 -16616.633,E2 -16616.633} C_VEL
LIN {X 0,Y 294.054,Z 255.402,A -85,B 0,C 180,E1 -16620.663,E2 -16620.663} C_VEL
LIN {X 0,Y 295.648,Z 263.887,A -85,B 0,C 180,E1 -16623.344,E2 -16623.344} C_VEL
LIN {X 0,Y 297.539,Z 270.335,A -85,B 0,C 180,E1 -16623.678,E2 -16623.678} C_VEL
LIN {X 0,Y 302.455,Z 301.777,A -85,B 0,C 180,E1 -16624.914,E2 -16624.914} C_VEL
LIN {X 0,Y 303.114,Z 307.67,A -85,B 0,C 180,E1 -16625.121,E2 -16625.121} C_VEL
LIN {X 0,Y 301.277,Z 372.831,A -85,B 0,C 180,E1 -16626.728,E2 -16626.728} C_VEL
LIN {X 0,Y 300.435,Z 385.706,A -85,B 0,C 180,E1 -16627.296,E2 -16627.296} C_VEL
LIN {X 0,Y 299.231,Z 398.261,A -85,B 0,C 180,E1 -16628.109,E2 -16628.109} C_VEL
LIN {X 0,Y 298.026,Z 409.485,A -85,B 0,C 180,E1 -16629.104,E2 -16629.104} C_VEL
LIN {X 0,Y 296.462,Z 421.131,A -85,B 0,C 180,E1 -16630.437,E2 -16630.437} C_VEL
LIN {X 0,Y 294.92,Z 431.622,A -85,B 0,C 180,E1 -16631.954,E2 -16631.954} C_VEL
LIN {X 0,Y 293.658,Z 441.07,A -85,B 0,C 180,E1 -16633.668,E2 -16633.668} C_VEL
LIN {X 0,Y 292.216,Z 450.176,A -85,B 0,C 180,E1 -16635.729,E2 -16635.729} C_VEL
LIN {X 0,Y 291.001,Z 457.501,A -85,B 0,C 180,E1 -16637.8,E2 -16637.8} C_VEL
LIN {X 0,Y 290.373,Z 462.454,A -85,B 0,C 180,E1 -16639.542,E2 -16639.542} C_VEL
LIN {X 0,Y 289.847,Z 467.255,A -85,B 0,C 180,E1 -16641.635,E2 -16641.635} C_VEL
LIN {X 0,Y 289.524,Z 470.917,A -85,B 0,C 180,E1 -16643.729,E2 -16643.729} C_VEL
LIN {X 0,Y 289.43,Z 473.549,A -85,B 0,C 180,E1 -16645.823,E2 -16645.823} C_VEL
LIN {X 0,Y 289.438,Z 474.782,A -85,B 0,C 180,E1 -16647.217,E2 -16647.217} C_VEL
LIN {X 0,Y 289.415,Z 475.585,A -85,B 0,C 180,E1 -16648.609,E2 -16648.609} C_VEL
LIN {X 0,Y 289.435,Z 475.961,A -85,B 0,C 180,E1 -16650,E2 -16650} C_VEL
LIN {X 0,Y 289.407,Z 475.945,A -85,B 0,C 180,E1 -16651.392,E2 -16651.392} C_VEL
LIN {X 0,Y 289.43,Z 475.542,A -85,B 0,C 180,E1 -16652.784,E2 -16652.784} C_VEL
LIN {X 0,Y 289.428,Z 473.673,A -85,B 0,C 180,E1 -16655.388,E2 -16655.388} C_VEL
LIN {X 0,Y 289.727,Z 470.84,A -85,B 0,C 180,E1 -16657.667,E2 -16657.667} C_VEL
LIN {X 0,Y 290.252,Z 467.193,A -85,B 0,C 180,E1 -16659.759,E2 -16659.759} C_VEL
LIN {X 0,Y 291.03,Z 462.44,A -85,B 0,C 180,E1 -16661.845,E2 -16661.845} C_VEL
LIN {X 0,Y 292.186,Z 456.451,A -85,B 0,C 180,E1 -16663.918,E2 -16663.918} C_VEL
LIN {X 0,Y 293.739,Z 449.008,A -85,B 0,C 180,E1 -16665.971,E2 -16665.971} C_VEL
LIN {X 0,Y 295.39,Z 439.778,A -85,B 0,C 180,E1 -16668.017,E2 -16668.017} C_VEL
LIN {X 0,Y 297.34,Z 429.143,A -85,B 0,C 180,E1 -16669.863,E2 -16669.863} C_VEL
LIN {X 0,Y 299.331,Z 418.328,A -85,B 0,C 180,E1 -16671.341,E2 -16671.341} C_VEL
LIN {X 0,Y 300.913,Z 407.806,A -85,B 0,C 180,E1 -16672.485,E2 -16672.485} C_VEL
LIN {X 0,Y 302.606,Z 395.192,A -85,B 0,C 180,E1 -16673.527,E2 -16673.527} C_VEL
LIN {X 0,Y 303.844,Z 382.674,A -85,B 0,C 180,E1 -16674.286,E2 -16674.286} C_VEL
LIN {X 0,Y 304.767,Z 369.713,A -85,B 0,C 180,E1 -16674.794,E2 -16674.794} C_VEL
LIN {X 0,Y 306.605,Z 306.949,A -85,B 0,C 180,E1 -16676.347,E2 -16676.347} C_VEL
LIN {X 0,Y 303.273,Z 285.665,A -85,B 0,C 180,E1 -16677.299,E2 -16677.299} C_VEL
LIN {X 0,Y 300.751,Z 273.896,A -85,B 0,C 180,E1 -16677.918,E2 -16677.918} C_VEL
LIN {X 0,Y 295.977,Z 262.565,A -85,B 0,C 180,E1 -16678.834,E2 -16678.834} C_VEL
LIN {X 0,Y 293.665,Z 252.287,A -85,B 0,C 180,E1 -16682.345,E2 -16682.345} C_VEL
LIN {X 0,Y 291.389,Z 243.189,A -85,B 0,C 180,E1 -16685.688,E2 -16685.688} C_VEL
LIN {X 0,Y 291.382,Z 243.188,A -85,B 0,C 180,E1 -16689.482,E2 -16689.482} C_VEL
LIN {X 0,Y 291.31,Z 243.202,A -85,B 0,C 180,E1 -16693.634,E2 -16693.634} C_VEL
LIN {X 0,Y 291.319,Z 243.194,A -85,B 0,C 180,E1 -16697.507,E2 -16697.507} C_VEL
LIN {X 0,Y 291.353,Z 243.188,A -85,B 0,C 180,E1 -16701.158,E2 -16701.158} C_VEL
LIN {X 0,Y 291.361,Z 243.185,A -85,B 0,C 180,E1 -16704.626,E2 -16704.626} C_VEL
LIN {X 0,Y 291.37,Z 243.184,A -85,B 0,C 180,E1 -16707.95,E2 -16707.95} C_VEL
LIN {X 0,Y 291.378,Z 243.188,A -85,B 0,C 180,E1 -16711.158,E2 -16711.158} C_VEL
LIN {X 0,Y 291.416,Z 243.183,A -85,B 0,C 180,E1 -16714.272,E2 -16714.272} C_VEL
LIN {X 0,Y 291.381,Z 243.181,A -85,B 0,C 180,E1 -16717.3,E2 -16717.3} C_VEL
LIN {X 0,Y 291.458,Z 243.177,A -85,B 0,C 180,E1 -16720.27,E2 -16720.27} C_VEL
LIN {X 0,Y 291.555,Z 243.164,A -85,B 0,C 180,E1 -16724.624,E2 -16724.624} C_VEL
LIN {X 0,Y 291.537,Z 243.168,A -85,B 0,C 180,E1 -16728.881,E2 -16728.881} C_VEL
LIN {X 0,Y 291.706,Z 243.145,A -85,B 0,C 180,E1 -16731.688,E2 -16731.688} C_VEL
LIN {X 0,Y 291.628,Z 243.151,A -85,B 0,C 180,E1 -16734.468,E2 -16734.468} C_VEL
LIN {X 0,Y 291.888,Z 243.121,A -85,B 0,C 180,E1 -16738.62,E2 -16738.62} C_VEL
LIN {X 0,Y 291.889,Z 243.126,A -85,B 0,C 180,E1 -16741.38,E2 -16741.38} C_VEL
LIN {X 0,Y 291.746,Z 243.14,A -85,B 0,C 180,E1 -16746.918,E2 -16746.918} C_VEL
LIN {X 0,Y 291.629,Z 243.158,A -85,B 0,C 180,E1 -16749.712,E2 -16749.712} C_VEL
LIN {X 0,Y 291.522,Z 243.172,A -85,B 0,C 180,E1 -16753.95,E2 -16753.95} C_VEL
LIN {X 0,Y 291.487,Z 243.178,A -85,B 0,C 180,E1 -16756.818,E2 -16756.818} C_VEL
LIN {X 0,Y 291.451,Z 243.181,A -85,B 0,C 180,E1 -16759.875,E2 -16759.875} C_VEL
LIN {X 0,Y 291.366,Z 243.19,A -85,B 0,C 180,E1 -16764.208,E2 -16764.208} C_VEL
LIN {X 0,Y 291.362,Z 243.193,A -85,B 0,C 180,E1 -16767.278,E2 -16767.278} C_VEL
LIN {X 0,Y 291.322,Z 243.196,A -85,B 0,C 180,E1 -16770.439,E2 -16770.439} C_VEL
LIN {X 0,Y 291.423,Z 243.375,A -85,B 0,C 180,E1 -16773.59,E2 -16773.59} C_VEL
LIN {X 0,Y 293.029,Z 249.626,A -85,B 0,C 180,E1 -16775.881,E2 -16775.881} C_VEL
LIN {X 0,Y 301.152,Z 266.453,A -85,B 0,C 180,E1 -16777.356,E2 -16777.356} C_VEL
LIN {X 0,Y 306.59,Z 279.839,A -85,B 0,C 180,E1 -16778.343,E2 -16778.343} C_VEL
LIN {X 0,Y 307.373,Z 285.185,A -85,B 0,C 180,E1 -16778.576,E2 -16778.576} C_VEL
LIN {X 0,Y 304.87,Z 357.741,A -85,B 0,C 180,E1 -16780.361,E2 -16780.361} C_VEL
LIN {X 0,Y 303.924,Z 371.651,A -85,B 0,C 180,E1 -16780.993,E2 -16780.993} C_VEL
LIN {X 0,Y 302.796,Z 383.461,A -85,B 0,C 180,E1 -16781.787,E2 -16781.787} C_VEL
LIN {X 0,Y 301.365,Z 395.196,A -85,B 0,C 180,E1 -16782.851,E2 -16782.851} C_VEL
LIN {X 0,Y 299.766,Z 405.816,A -85,B 0,C 180,E1 -16784.079,E2 -16784.079} C_VEL
LIN {X 0,Y 297.914,Z 416.694,A -85,B 0,C 180,E1 -16785.663,E2 -16785.663} C_VEL
LIN {X 0,Y 296.121,Z 425.999,A -85,B 0,C 180,E1 -16787.37,E2 -16787.37} C_VEL
LIN {X 0,Y 294.345,Z 434.881,A -85,B 0,C 180,E1 -16789.41,E2 -16789.41} C_VEL
LIN {X 0,Y 292.925,Z 441.825,A -85,B 0,C 180,E1 -16791.406,E2 -16791.406} C_VEL
LIN {X 0,Y 291.986,Z 446.351,A -85,B 0,C 180,E1 -16793.005,E2 -16793.005} C_VEL
LIN {X 0,Y 290.964,Z 451.383,A -85,B 0,C 180,E1 -16795.21,E2 -16795.21} C_VEL
LIN {X 0,Y 290.14,Z 455.719,A -85,B 0,C 180,E1 -16797.798,E2 -16797.798} C_VEL
LIN {X 0,Y 289.742,Z 457.576,A -85,B 0,C 180,E1 -16799.378,E2 -16799.378} C_VEL
LIN {X 0,Y 289.467,Z 458.932,A -85,B 0,C 180,E1 -16800.949,E2 -16800.949} C_VEL
LIN {X 0,Y 289.262,Z 459.721,A -85,B 0,C 180,E1 -16802.508,E2 -16802.508} C_VEL
LIN {X 0,Y 289.176,Z 460.038,A -85,B 0,C 180,E1 -16804.058,E2 -16804.058} C_VEL
LIN {X 0,Y 289.1,Z 459.875,A -85,B 0,C 180,E1 -16805.59,E2 -16805.59} C_VEL
LIN {X 0,Y 289.171,Z 459.004,A -85,B 0,C 180,E1 -16807.452,E2 -16807.452} C_VEL
LIN {X 0,Y 289.545,Z 456.477,A -85,B 0,C 180,E1 -16810.134,E2 -16810.134} C_VEL
LIN {X 0,Y 290.054,Z 453.142,A -85,B 0,C 180,E1 -16812.37,E2 -16812.37} C_VEL
LIN {X 0,Y 290.626,Z 448.66,A -85,B 0,C 180,E1 -16814.573,E2 -16814.573} C_VEL
LIN {X 0,Y 291.502,Z 442.878,A -85,B 0,C 180,E1 -16816.759,E2 -16816.759} C_VEL
LIN {X 0,Y 292.637,Z 435.624,A -85,B 0,C 180,E1 -16818.923,E2 -16818.923} C_VEL
LIN {X 0,Y 293.846,Z 428.145,A -85,B 0,C 180,E1 -16820.709,E2 -16820.709} C_VEL
LIN {X 0,Y 295.361,Z 418.039,A -85,B 0,C 180,E1 -16822.652,E2 -16822.652} C_VEL
LIN {X 0,Y 296.915,Z 407.036,A -85,B 0,C 180,E1 -16824.33,E2 -16824.33} C_VEL
LIN {X 0,Y 298.358,Z 396.327,A -85,B 0,C 180,E1 -16825.609,E2 -16825.609} C_VEL
LIN {X 0,Y 299.7,Z 383.486,A -85,B 0,C 180,E1 -16826.807,E2 -16826.807} C_VEL
LIN {X 0,Y 300.639,Z 371.131,A -85,B 0,C 180,E1 -16827.655,E2 -16827.655} C_VEL
LIN {X 0,Y 301.427,Z 357.344,A -85,B 0,C 180,E1 -16828.288,E2 -16828.288} C_VEL
LIN {X 0,Y 302.762,Z 313.958,A -85,B 0,C 180,E1 -16829.368,E2 -16829.368} C_VEL
LIN {X 0,Y 303.552,Z 282,A -85,B 0,C 180,E1 -16830.145,E2 -16830.145} C_VEL
LIN {X 0,Y 301.382,Z 271.509,A -85,B 0,C 180,E1 -16830.596,E2 -16830.596} C_VEL
LIN {X 0,Y 293.872,Z 251.379,A -85,B 0,C 180,E1 -16831.775,E2 -16831.775} C_VEL
LIN {X 0,Y 293.01,Z 248.913,A -85,B 0,C 180,E1 -16831.946,E2 -16831.946} C_VEL
LIN {X 0,Y 291.53,Z 243.177,A -85,B 0,C 180,E1 -16834.061,E2 -16834.061} C_VEL
LIN {X 0,Y 291.69,Z 243.153,A -85,B 0,C 180,E1 -16836.919,E2 -16836.919} C_VEL
LIN {X 0,Y 291.571,Z 243.166,A -85,B 0,C 180,E1 -16839.714,E2 -16839.714} C_VEL
LIN {X 0,Y 291.524,Z 243.175,A -85,B 0,C 180,E1 -16843.95,E2 -16843.95} C_VEL
LIN {X 0,Y 291.489,Z 243.176,A -85,B 0,C 180,E1 -16846.817,E2 -16846.817} C_VEL
LIN {X 0,Y 291.453,Z 243.184,A -85,B 0,C 180,E1 -16849.874,E2 -16849.874} C_VEL
LIN {X 0,Y 291.368,Z 243.191,A -85,B 0,C 180,E1 -16854.208,E2 -16854.208} C_VEL
LIN {X 0,Y 291.36,Z 243.189,A -85,B 0,C 180,E1 -16857.277,E2 -16857.277} C_VEL
LIN {X 0,Y 291.321,Z 243.195,A -85,B 0,C 180,E1 -16860.438,E2 -16860.438} C_VEL
LIN {X 0,Y 291.344,Z 243.195,A -85,B 0,C 180,E1 -16863.698,E2 -16863.698} C_VEL
LIN {X 0,Y 291.381,Z 243.185,A -85,B 0,C 180,E1 -16867.255,E2 -16867.255} C_VEL
LIN {X 0,Y 291.333,Z 243.193,A -85,B 0,C 180,E1 -16870.642,E2 -16870.642} C_VEL
LIN {X 0,Y 291.29,Z 243.194,A -85,B 0,C 180,E1 -16874.401,E2 -16874.401} C_VEL
LIN {X 0,Y 291.325,Z 243.195,A -85,B 0,C 180,E1 -16878.404,E2 -16878.404} C_VEL
LIN {X 0,Y 291.362,Z 243.188,A -85,B 0,C 180,E1 -16881.159,E2 -16881.159} C_VEL
LIN {X 0,Y 291.36,Z 243.182,A -85,B 0,C 180,E1 -16884.626,E2 -16884.626} C_VEL
LIN {X 0,Y 291.369,Z 243.19,A -85,B 0,C 180,E1 -16887.95,E2 -16887.95} C_VEL
LIN {X 0,Y 291.376,Z 243.187,A -85,B 0,C 180,E1 -16891.157,E2 -16891.157} C_VEL
LIN {X 0,Y 291.434,Z 243.176,A -85,B 0,C 180,E1 -16893.218,E2 -16893.218} C_VEL
LIN {X 0,Y 290.707,Z 243.265,A -85,B 0,C 180,E1 -16894.371,E2 -16894.371} C_VEL
LIN {X 0,Y 287.797,Z 243.625,A -85,B 0,C 180,E1 -16896.248,E2 -16896.248} C_VEL
LIN {X 0,Y 285.389,Z 243.926,A -85,B 0,C 180,E1 -16897.772,E2 -16897.772} C_VEL
LIN {X 0,Y 284.401,Z 244.052,A -85,B 0,C 180,E1 -16898.953,E2 -16898.953} C_VEL
LIN {X 0,Y 284.344,Z 244.059,A -85,B 0,C 180,E1 -16899.353,E2 -16899.353} C_VEL
LIN {X 0,Y 284.423,Z 244.053,A -85,B 0,C 180,E1 -16902.751,E2 -16902.751} C_VEL
LIN {X 0,Y 284.479,Z 244.046,A -85,B 0,C 180,E1 -16905.697,E2 -16905.697} C_VEL
LIN {X 0,Y 284.664,Z 244.017,A -85,B 0,C 180,E1 -16910.946,E2 -16910.946} C_VEL
LIN {X 0,Y 284.599,Z 244.035,A -85,B 0,C 180,E1 -16914.331,E2 -16914.331} C_VEL
LIN {X 0,Y 284.854,Z 243.997,A -85,B 0,C 180,E1 -16918.586,E2 -16918.586} C_VEL
LIN {X 0,Y 284.853,Z 243.99,A -85,B 0,C 180,E1 -16921.414,E2 -16921.414} C_VEL
LIN {X 0,Y 284.696,Z 244.019,A -85,B 0,C 180,E1 -16927.09,E2 -16927.09} C_VEL
LIN {X 0,Y 284.564,Z 244.038,A -85,B 0,C 180,E1 -16929.955,E2 -16929.955} C_VEL
LIN {X 0,Y 284.479,Z 244.041,A -85,B 0,C 180,E1 -16934.303,E2 -16934.303} C_VEL
LIN {X 0,Y 284.423,Z 244.053,A -85,B 0,C 180,E1 -16937.248,E2 -16937.248} C_VEL
LIN {X 0,Y 284.377,Z 244.062,A -85,B 0,C 180,E1 -16940.242,E2 -16940.242} C_VEL
LIN {X 0,Y 284.368,Z 244.06,A -85,B 0,C 180,E1 -16943.876,E2 -16943.876} C_VEL
LIN {X 0,Y 284.395,Z 244.056,A -85,B 0,C 180,E1 -16947.174,E2 -16947.174} C_VEL
LIN {X 0,Y 284.294,Z 244.07,A -85,B 0,C 180,E1 -16951.275,E2 -16951.275} C_VEL
LIN {X 0,Y 284.339,Z 244.064,A -85,B 0,C 180,E1 -16955.348,E2 -16955.348} C_VEL
LIN {X 0,Y 284.31,Z 244.069,A -85,B 0,C 180,E1 -16958.169,E2 -16958.169} C_VEL
LIN {X 0,Y 284.268,Z 244.072,A -85,B 0,C 180,E1 -16962.125,E2 -16962.125} C_VEL
LIN {X 0,Y 284.254,Z 244.079,A -85,B 0,C 180,E1 -16966.19,E2 -16966.19} C_VEL
LIN {X 0,Y 284.312,Z 244.07,A -85,B 0,C 180,E1 -16970.023,E2 -16970.023} C_VEL
LIN {X 0,Y 284.35,Z 244.066,A -85,B 0,C 180,E1 -16973.617,E2 -16973.617} C_VEL
LIN {X 0,Y 284.401,Z 244.225,A -85,B 0,C 180,E1 -16976.168,E2 -16976.168} C_VEL
LIN {X 0,Y 286.725,Z 254.895,A -85,B 0,C 180,E1 -16979.839,E2 -16979.839} C_VEL
LIN {X 0,Y 288.458,Z 263.655,A -85,B 0,C 180,E1 -16982.712,E2 -16982.712} C_VEL
LIN {X 0,Y 291.175,Z 272.228,A -85,B 0,C 180,E1 -16983.189,E2 -16983.189} C_VEL
LIN {X 0,Y 296.375,Z 306.341,A -85,B 0,C 180,E1 -16984.554,E2 -16984.554} C_VEL
LIN {X 0,Y 295.695,Z 339.156,A -85,B 0,C 180,E1 -16985.38,E2 -16985.38} C_VEL
LIN {X 0,Y 294.701,Z 372.122,A -85,B 0,C 180,E1 -16986.223,E2 -16986.223} C_VEL
LIN {X 0,Y 293.787,Z 385.152,A -85,B 0,C 180,E1 -16986.799,E2 -16986.799} C_VEL
LIN {X 0,Y 292.661,Z 397.247,A -85,B 0,C 180,E1 -16987.591,E2 -16987.591} C_VEL
LIN {X 0,Y 291.364,Z 408.693,A -85,B 0,C 180,E1 -16988.603,E2 -16988.603} C_VEL
LIN {X 0,Y 289.774,Z 420.464,A -85,B 0,C 180,E1 -16989.966,E2 -16989.966} C_VEL
LIN {X 0,Y 288.079,Z 431.029,A -85,B 0,C 180,E1 -16991.51,E2 -16991.51} C_VEL
LIN {X 0,Y 286.789,Z 440.572,A -85,B 0,C 180,E1 -16993.266,E2 -16993.266} C_VEL
LIN {X 0,Y 285.314,Z 449.734,A -85,B 0,C 180,E1 -16995.376,E2 -16995.376} C_VEL
LIN {X 0,Y 284.036,Z 457.103,A -85,B 0,C 180,E1 -16997.497,E2 -16997.497} C_VEL
LIN {X 0,Y 283.366,Z 462.095,A -85,B 0,C 180,E1 -16999.28,E2 -16999.28} C_VEL
LIN {X 0,Y 282.795,Z 466.931,A -85,B 0,C 180,E1 -17001.425,E2 -17001.425} C_VEL
LIN {X 0,Y 282.445,Z 470.626,A -85,B 0,C 180,E1 -17003.571,E2 -17003.571} C_VEL
LIN {X 0,Y 282.337,Z 473.288,A -85,B 0,C 180,E1 -17005.718,E2 -17005.718} C_VEL
LIN {X 0,Y 282.345,Z 474.536,A -85,B 0,C 180,E1 -17007.147,E2 -17007.147} C_VEL
LIN {X 0,Y 282.338,Z 475.366,A -85,B 0,C 180,E1 -17008.574,E2 -17008.574} C_VEL
LIN {X 0,Y 282.355,Z 475.757,A -85,B 0,C 180,E1 -17010,E2 -17010} C_VEL
LIN {X 0,Y 282.33,Z 475.755,A -85,B 0,C 180,E1 -17011.427,E2 -17011.427} C_VEL
LIN {X 0,Y 282.336,Z 475.365,A -85,B 0,C 180,E1 -17012.854,E2 -17012.854} C_VEL
LIN {X 0,Y 282.337,Z 473.734,A -85,B 0,C 180,E1 -17015.32,E2 -17015.32} C_VEL
LIN {X 0,Y 282.684,Z 470.737,A -85,B 0,C 180,E1 -17017.859,E2 -17017.859} C_VEL
LIN {X 0,Y 283.219,Z 467.127,A -85,B 0,C 180,E1 -17020.003,E2 -17020.003} C_VEL
LIN {X 0,Y 284.05,Z 462.417,A -85,B 0,C 180,E1 -17022.141,E2 -17022.141} C_VEL
LIN {X 0,Y 285.286,Z 456.468,A -85,B 0,C 180,E1 -17024.262,E2 -17024.262} C_VEL
LIN {X 0,Y 286.9,Z 449.07,A -85,B 0,C 180,E1 -17026.362,E2 -17026.362} C_VEL
LIN {X 0,Y 288.647,Z 439.914,A -85,B 0,C 180,E1 -17028.453,E2 -17028.453} C_VEL
LIN {X 0,Y 290.692,Z 429.35,A -85,B 0,C 180,E1 -17030.337,E2 -17030.337} C_VEL
LIN {X 0,Y 292.75,Z 418.625,A -85,B 0,C 180,E1 -17031.846,E2 -17031.846} C_VEL
LIN {X 0,Y 294.399,Z 408.256,A -85,B 0,C 180,E1 -17033.011,E2 -17033.011} C_VEL
LIN {X 0,Y 296.153,Z 395.848,A -85,B 0,C 180,E1 -17034.072,E2 -17034.072} C_VEL
LIN {X 0,Y 297.493,Z 382.907,A -85,B 0,C 180,E1 -17034.885,E2 -17034.885} C_VEL
LIN {X 0,Y 298.46,Z 370.438,A -85,B 0,C 180,E1 -17035.4,E2 -17035.4} C_VEL
LIN {X 0,Y 300.432,Z 308.103,A -85,B 0,C 180,E1 -17036.976,E2 -17036.976} C_VEL
LIN {X 0,Y 297.25,Z 287.455,A -85,B 0,C 180,E1 -17037.931,E2 -17037.931} C_VEL
LIN {X 0,Y 295.007,Z 276.861,A -85,B 0,C 180,E1 -17038.504,E2 -17038.504} C_VEL
LIN {X 0,Y 289.941,Z 265.281,A -85,B 0,C 180,E1 -17039.48,E2 -17039.48} C_VEL
LIN {X 0,Y 288.699,Z 262.253,A -85,B 0,C 180,E1 -17039.773,E2 -17039.773} C_VEL
LIN {X 0,Y 286.382,Z 251.938,A -85,B 0,C 180,E1 -17043.448,E2 -17043.448} C_VEL
LIN {X 0,Y 284.337,Z 244.067,A -85,B 0,C 180,E1 -17046.495,E2 -17046.495} C_VEL
LIN {X 0,Y 284.306,Z 244.067,A -85,B 0,C 180,E1 -17049.995,E2 -17049.995} C_VEL
LIN {X 0,Y 284.246,Z 244.08,A -85,B 0,C 180,E1 -17054.19,E2 -17054.19} C_VEL
LIN {X 0,Y 284.272,Z 244.069,A -85,B 0,C 180,E1 -17058.124,E2 -17058.124} C_VEL
LIN {X 0,Y 284.322,Z 244.066,A -85,B 0,C 180,E1 -17062.278,E2 -17062.278} C_VEL
LIN {X 0,Y 284.309,Z 244.064,A -85,B 0,C 180,E1 -17065.351,E2 -17065.351} C_VEL
LIN {X 0,Y 284.293,Z 244.063,A -85,B 0,C 180,E1 -17068.725,E2 -17068.725} C_VEL
LIN {X 0,Y 284.396,Z 244.05,A -85,B 0,C 180,E1 -17072.827,E2 -17072.827} C_VEL
LIN {X 0,Y 284.366,Z 244.054,A -85,B 0,C 180,E1 -17076.707,E2 -17076.707} C_VEL
LIN {X 0,Y 284.403,Z 244.048,A -85,B 0,C 180,E1 -17081.262,E2 -17081.262} C_VEL
LIN {X 0,Y 284.492,Z 244.046,A -85,B 0,C 180,E1 -17084.459,E2 -17084.459} C_VEL
LIN {X 0,Y 284.488,Z 244.048,A -85,B 0,C 180,E1 -17088.602,E2 -17088.602} C_VEL
LIN {X 0,Y 284.657,Z 244.02,A -85,B 0,C 180,E1 -17091.481,E2 -17091.481} C_VEL
LIN {X 0,Y 284.598,Z 244.027,A -85,B 0,C 180,E1 -17094.331,E2 -17094.331} C_VEL
LIN {X 0,Y 284.855,Z 243.997,A -85,B 0,C 180,E1 -17098.586,E2 -17098.586} C_VEL
LIN {X 0,Y 284.855,Z 244.002,A -85,B 0,C 180,E1 -17101.414,E2 -17101.414} C_VEL
LIN {X 0,Y 284.698,Z 244.017,A -85,B 0,C 180,E1 -17107.09,E2 -17107.09} C_VEL
LIN {X 0,Y 284.567,Z 244.038,A -85,B 0,C 180,E1 -17109.955,E2 -17109.955} C_VEL
LIN {X 0,Y 284.482,Z 244.048,A -85,B 0,C 180,E1 -17114.303,E2 -17114.303} C_VEL
LIN {X 0,Y 284.426,Z 244.055,A -85,B 0,C 180,E1 -17117.249,E2 -17117.249} C_VEL
LIN {X 0,Y 284.378,Z 244.063,A -85,B 0,C 180,E1 -17120.242,E2 -17120.242} C_VEL
LIN {X 0,Y 284.316,Z 244.073,A -85,B 0,C 180,E1 -17124.849,E2 -17124.849} C_VEL
LIN {X 0,Y 284.291,Z 244.067,A -85,B 0,C 180,E1 -17128.015,E2 -17128.015} C_VEL
LIN {X 0,Y 284.287,Z 244.072,A -85,B 0,C 180,E1 -17131.276,E2 -17131.276} C_VEL
LIN {X 0,Y 284.338,Z 244.116,A -85,B 0,C 180,E1 -17132.755,E2 -17132.755} C_VEL
LIN {X 0,Y 285.845,Z 249.825,A -85,B 0,C 180,E1 -17134.943,E2 -17134.943} C_VEL
LIN {X 0,Y 294.593,Z 267.562,A -85,B 0,C 180,E1 -17136.614,E2 -17136.614} C_VEL
LIN {X 0,Y 300.607,Z 282.173,A -85,B 0,C 180,E1 -17137.744,E2 -17137.744} C_VEL
LIN {X 0,Y 301.226,Z 285.911,A -85,B 0,C 180,E1 -17137.921,E2 -17137.921} C_VEL
LIN {X 0,Y 298.658,Z 357.539,A -85,B 0,C 180,E1 -17139.718,E2 -17139.718} C_VEL
LIN {X 0,Y 297.703,Z 370.858,A -85,B 0,C 180,E1 -17140.32,E2 -17140.32} C_VEL
LIN {X 0,Y 296.418,Z 383.716,A -85,B 0,C 180,E1 -17141.187,E2 -17141.187} C_VEL
LIN {X 0,Y 294.812,Z 396.193,A -85,B 0,C 180,E1 -17142.353,E2 -17142.353} C_VEL
LIN {X 0,Y 293.016,Z 407.624,A -85,B 0,C 180,E1 -17143.735,E2 -17143.735} C_VEL
LIN {X 0,Y 291.12,Z 417.97,A -85,B 0,C 180,E1 -17145.323,E2 -17145.323} C_VEL
LIN {X 0,Y 289.209,Z 427.349,A -85,B 0,C 180,E1 -17147.124,E2 -17147.124} C_VEL
LIN {X 0,Y 287.486,Z 435.593,A -85,B 0,C 180,E1 -17149.095,E2 -17149.095} C_VEL
LIN {X 0,Y 285.963,Z 442.609,A -85,B 0,C 180,E1 -17151.194,E2 -17151.194} C_VEL
LIN {X 0,Y 284.52,Z 448.96,A -85,B 0,C 180,E1 -17153.642,E2 -17153.642} C_VEL
LIN {X 0,Y 283.538,Z 453.759,A -85,B 0,C 180,E1 -17156.103,E2 -17156.103} C_VEL
LIN {X 0,Y 282.842,Z 457.146,A -85,B 0,C 180,E1 -17158.547,E2 -17158.547} C_VEL
LIN {X 0,Y 282.422,Z 458.974,A -85,B 0,C 180,E1 -17160.572,E2 -17160.572} C_VEL
LIN {X 0,Y 282.116,Z 460.177,A -85,B 0,C 180,E1 -17163.358,E2 -17163.358} C_VEL
LIN {X 0,Y 282.028,Z 460.179,A -85,B 0,C 180,E1 -17164.936,E2 -17164.936} C_VEL
LIN {X 0,Y 282.072,Z 459.343,A -85,B 0,C 180,E1 -17167.203,E2 -17167.203} C_VEL
LIN {X 0,Y 282.349,Z 457.347,A -85,B 0,C 180,E1 -17169.606,E2 -17169.606} C_VEL
LIN {X 0,Y 282.864,Z 454.303,A -85,B 0,C 180,E1 -17171.906,E2 -17171.906} C_VEL
LIN {X 0,Y 283.402,Z 450.145,A -85,B 0,C 180,E1 -17174.17,E2 -17174.17} C_VEL
LIN {X 0,Y 284.215,Z 444.72,A -85,B 0,C 180,E1 -17176.413,E2 -17176.413} C_VEL
LIN {X 0,Y 285.362,Z 437.814,A -85,B 0,C 180,E1 -17178.637,E2 -17178.637} C_VEL
LIN {X 0,Y 286.797,Z 429.205,A -85,B 0,C 180,E1 -17180.835,E2 -17180.835} C_VEL
LIN {X 0,Y 288.232,Z 420.317,A -85,B 0,C 180,E1 -17182.645,E2 -17182.645} C_VEL
LIN {X 0,Y 289.631,Z 410.873,A -85,B 0,C 180,E1 -17184.204,E2 -17184.204} C_VEL
LIN {X 0,Y 291.221,Z 399.722,A -85,B 0,C 180,E1 -17185.675,E2 -17185.675} C_VEL
LIN {X 0,Y 292.543,Z 387.917,A -85,B 0,C 180,E1 -17186.901,E2 -17186.901} C_VEL
LIN {X 0,Y 293.681,Z 375.571,A -85,B 0,C 180,E1 -17187.857,E2 -17187.857} C_VEL
LIN {X 0,Y 294.552,Z 363.058,A -85,B 0,C 180,E1 -17188.547,E2 -17188.547} C_VEL
LIN {X 0,Y 295.117,Z 350.367,A -85,B 0,C 180,E1 -17188.989,E2 -17188.989} C_VEL
LIN {X 0,Y 297.019,Z 283.192,A -85,B 0,C 180,E1 -17190.641,E2 -17190.641} C_VEL
LIN {X 0,Y 295.027,Z 273.63,A -85,B 0,C 180,E1 -17191.066,E2 -17191.066} C_VEL
LIN {X 0,Y 287.977,Z 254.679,A -85,B 0,C 180,E1 -17192.206,E2 -17192.206} C_VEL
LIN {X 0,Y 285.799,Z 249.139,A -85,B 0,C 180,E1 -17192.581,E2 -17192.581} C_VEL
LIN {X 0,Y 284.5,Z 244.051,A -85,B 0,C 180,E1 -17194.516,E2 -17194.516} C_VEL
LIN {X 0,Y 284.645,Z 244.03,A -85,B 0,C 180,E1 -17197.091,E2 -17197.091} C_VEL
LIN {X 0,Y 284.516,Z 244.044,A -85,B 0,C 180,E1 -17199.957,E2 -17199.957} C_VEL
LIN {X 0,Y 284.484,Z 244.05,A -85,B 0,C 180,E1 -17204.302,E2 -17204.302} C_VEL
LIN {X 0,Y 284.427,Z 244.057,A -85,B 0,C 180,E1 -17207.248,E2 -17207.248} C_VEL
LIN {X 0,Y 284.379,Z 244.062,A -85,B 0,C 180,E1 -17210.242,E2 -17210.242} C_VEL
LIN {X 0,Y 284.327,Z 244.066,A -85,B 0,C 180,E1 -17213.855,E2 -17213.855} C_VEL
LIN {X 0,Y 284.29,Z 244.069,A -85,B 0,C 180,E1 -17218.015,E2 -17218.015} C_VEL
LIN {X 0,Y 284.286,Z 244.071,A -85,B 0,C 180,E1 -17221.275,E2 -17221.275} C_VEL
LIN {X 0,Y 284.341,Z 244.06,A -85,B 0,C 180,E1 -17225.347,E2 -17225.347} C_VEL
LIN {X 0,Y 284.318,Z 244.07,A -85,B 0,C 180,E1 -17228.167,E2 -17228.167} C_VEL
LIN {X 0,Y 284.268,Z 244.071,A -85,B 0,C 180,E1 -17232.124,E2 -17232.124} C_VEL
LIN {X 0,Y 284.255,Z 244.076,A -85,B 0,C 180,E1 -17236.189,E2 -17236.189} C_VEL
LIN {X 0,Y 284.306,Z 244.071,A -85,B 0,C 180,E1 -17240.023,E2 -17240.023} C_VEL
LIN {X 0,Y 284.333,Z 244.06,A -85,B 0,C 180,E1 -17243.614,E2 -17243.614} C_VEL
LIN {X 0,Y 284.306,Z 244.065,A -85,B 0,C 180,E1 -17247.189,E2 -17247.189} C_VEL
LIN {X 0,Y 284.354,Z 244.064,A -85,B 0,C 180,E1 -17250.375,E2 -17250.375} C_VEL
LIN {X 0,Y 284.376,Z 244.057,A -85,B 0,C 180,E1 -17253.586,E2 -17253.586} C_VEL
LIN {X 0,Y 284.364,Z 244.051,A -85,B 0,C 180,E1 -17256.707,E2 -17256.707} C_VEL
LIN {X 0,Y 284.344,Z 244.059,A -85,B 0,C 180,E1 -17259.353,E2 -17259.353} C_VEL
LIN {X 0,Y 283.752,Z 244.139,A -85,B 0,C 180,E1 -17260.535,E2 -17260.535} C_VEL
LIN {X 0,Y 280.979,Z 244.489,A -85,B 0,C 180,E1 -17262.462,E2 -17262.462} C_VEL
LIN {X 0,Y 278.572,Z 244.786,A -85,B 0,C 180,E1 -17264.027,E2 -17264.027} C_VEL
LIN {X 0,Y 277.511,Z 244.912,A -85,B 0,C 180,E1 -17265.239,E2 -17265.239} C_VEL
LIN {X 0,Y 277.413,Z 244.921,A -85,B 0,C 180,E1 -17265.65,E2 -17265.65} C_VEL
LIN {X 0,Y 277.629,Z 244.893,A -85,B 0,C 180,E1 -17270.841,E2 -17270.841} C_VEL
LIN {X 0,Y 277.57,Z 244.91,A -85,B 0,C 180,E1 -17274.187,E2 -17274.187} C_VEL
LIN {X 0,Y 277.82,Z 244.873,A -85,B 0,C 180,E1 -17278.55,E2 -17278.55} C_VEL
LIN {X 0,Y 277.819,Z 244.865,A -85,B 0,C 180,E1 -17281.449,E2 -17281.449} C_VEL
LIN {X 0,Y 277.651,Z 244.897,A -85,B 0,C 180,E1 -17287.271,E2 -17287.271} C_VEL
LIN {X 0,Y 277.505,Z 244.916,A -85,B 0,C 180,E1 -17290.211,E2 -17290.211} C_VEL
LIN {X 0,Y 277.432,Z 244.921,A -85,B 0,C 180,E1 -17294.674,E2 -17294.674} C_VEL
LIN {X 0,Y 277.343,Z 244.935,A -85,B 0,C 180,E1 -17299.234,E2 -17299.234} C_VEL
LIN {X 0,Y 277.318,Z 244.94,A -85,B 0,C 180,E1 -17304.171,E2 -17304.171} C_VEL
LIN {X 0,Y 277.324,Z 244.937,A -85,B 0,C 180,E1 -17307.506,E2 -17307.506} C_VEL
LIN {X 0,Y 277.27,Z 244.949,A -85,B 0,C 180,E1 -17310.482,E2 -17310.482} C_VEL
LIN {X 0,Y 277.245,Z 244.947,A -85,B 0,C 180,E1 -17313.896,E2 -17313.896} C_VEL
LIN {X 0,Y 277.266,Z 244.944,A -85,B 0,C 180,E1 -17317.47,E2 -17317.47} C_VEL
LIN {X 0,Y 277.208,Z 244.95,A -85,B 0,C 180,E1 -17321.237,E2 -17321.237} C_VEL
LIN {X 0,Y 277.2,Z 244.955,A -85,B 0,C 180,E1 -17325.227,E2 -17325.227} C_VEL
LIN {X 0,Y 277.22,Z 244.954,A -85,B 0,C 180,E1 -17328.766,E2 -17328.766} C_VEL
LIN {X 0,Y 277.281,Z 244.948,A -85,B 0,C 180,E1 -17332.533,E2 -17332.533} C_VEL
LIN {X 0,Y 277.354,Z 245.135,A -85,B 0,C 180,E1 -17335.681,E2 -17335.681} C_VEL
LIN {X 0,Y 279.929,Z 256.967,A -85,B 0,C 180,E1 -17339.86,E2 -17339.86} C_VEL
LIN {X 0,Y 281.218,Z 263.459,A -85,B 0,C 180,E1 -17342.044,E2 -17342.044} C_VEL
LIN {X 0,Y 284.793,Z 273.859,A -85,B 0,C 180,E1 -17342.672,E2 -17342.672} C_VEL
LIN {X 0,Y 289.797,Z 307.013,A -85,B 0,C 180,E1 -17344.038,E2 -17344.038} C_VEL
LIN {X 0,Y 289.358,Z 331.856,A -85,B 0,C 180,E1 -17344.686,E2 -17344.686} C_VEL
LIN {X 0,Y 288.068,Z 372.264,A -85,B 0,C 180,E1 -17345.737,E2 -17345.737} C_VEL
LIN {X 0,Y 287.082,Z 385.943,A -85,B 0,C 180,E1 -17346.368,E2 -17346.368} C_VEL
LIN {X 0,Y 285.805,Z 398.319,A -85,B 0,C 180,E1 -17347.214,E2 -17347.214} C_VEL
LIN {X 0,Y 284.28,Z 411.014,A -85,B 0,C 180,E1 -17348.424,E2 -17348.424} C_VEL
LIN {X 0,Y 282.658,Z 422.319,A -85,B 0,C 180,E1 -17349.819,E2 -17349.819} C_VEL
LIN {X 0,Y 281.028,Z 432.497,A -85,B 0,C 180,E1 -17351.407,E2 -17351.407} C_VEL
LIN {X 0,Y 279.681,Z 441.688,A -85,B 0,C 180,E1 -17353.204,E2 -17353.204} C_VEL
LIN {X 0,Y 278.166,Z 450.631,A -85,B 0,C 180,E1 -17355.366,E2 -17355.366} C_VEL
LIN {X 0,Y 276.897,Z 457.788,A -85,B 0,C 180,E1 -17357.541,E2 -17357.541} C_VEL
LIN {X 0,Y 276.129,Z 463.492,A -85,B 0,C 180,E1 -17359.738,E2 -17359.738} C_VEL
LIN {X 0,Y 275.599,Z 467.97,A -85,B 0,C 180,E1 -17361.938,E2 -17361.938} C_VEL
LIN {X 0,Y 275.264,Z 472.052,A -85,B 0,C 180,E1 -17364.713,E2 -17364.713} C_VEL
LIN {X 0,Y 275.255,Z 474.286,A -85,B 0,C 180,E1 -17367.073,E2 -17367.073} C_VEL
LIN {X 0,Y 275.263,Z 475.142,A -85,B 0,C 180,E1 -17368.537,E2 -17368.537} C_VEL
LIN {X 0,Y 275.277,Z 475.553,A -85,B 0,C 180,E1 -17370,E2 -17370} C_VEL
LIN {X 0,Y 275.255,Z 475.566,A -85,B 0,C 180,E1 -17371.463,E2 -17371.463} C_VEL
LIN {X 0,Y 275.244,Z 475.19,A -85,B 0,C 180,E1 -17372.927,E2 -17372.927} C_VEL
LIN {X 0,Y 275.238,Z 473.773,A -85,B 0,C 180,E1 -17375.229,E2 -17375.229} C_VEL
LIN {X 0,Y 275.635,Z 470.644,A -85,B 0,C 180,E1 -17378.062,E2 -17378.062} C_VEL
LIN {X 0,Y 276.208,Z 467.068,A -85,B 0,C 180,E1 -17380.26,E2 -17380.26} C_VEL
LIN {X 0,Y 277.088,Z 462.394,A -85,B 0,C 180,E1 -17382.45,E2 -17382.45} C_VEL
LIN {X 0,Y 278.664,Z 455.36,A -85,B 0,C 180,E1 -17384.982,E2 -17384.982} C_VEL
LIN {X 0,Y 280.296,Z 447.77,A -85,B 0,C 180,E1 -17387.134,E2 -17387.134} C_VEL
LIN {X 0,Y 282.268,Z 438.286,A -85,B 0,C 180,E1 -17389.263,E2 -17389.263} C_VEL
LIN {X 0,Y 284.298,Z 428.518,A -85,B 0,C 180,E1 -17391.005,E2 -17391.005} C_VEL
LIN {X 0,Y 286.414,Z 417.667,A -85,B 0,C 180,E1 -17392.545,E2 -17392.545} C_VEL
LIN {X 0,Y 288.425,Z 405.336,A -85,B 0,C 180,E1 -17393.897,E2 -17393.897} C_VEL
LIN {X 0,Y 290.145,Z 393.299,A -85,B 0,C 180,E1 -17394.889,E2 -17394.889} C_VEL
LIN {X 0,Y 291.423,Z 380.959,A -85,B 0,C 180,E1 -17395.632,E2 -17395.632} C_VEL
LIN {X 0,Y 292.346,Z 367.94,A -85,B 0,C 180,E1 -17396.134,E2 -17396.134} C_VEL
LIN {X 0,Y 294.231,Z 308.57,A -85,B 0,C 180,E1 -17397.664,E2 -17397.664} C_VEL
LIN {X 0,Y 291.182,Z 288.81,A -85,B 0,C 180,E1 -17398.612,E2 -17398.612} C_VEL
LIN {X 0,Y 289.283,Z 279.659,A -85,B 0,C 180,E1 -17399.125,E2 -17399.125} C_VEL
LIN {X 0,Y 284.252,Z 268.21,A -85,B 0,C 180,E1 -17400.138,E2 -17400.138} C_VEL
LIN {X 0,Y 281.478,Z 261.962,A -85,B 0,C 180,E1 -17400.768,E2 -17400.768} C_VEL
LIN {X 0,Y 279.131,Z 251.903,A -85,B 0,C 180,E1 -17404.52,E2 -17404.52} C_VEL
LIN {X 0,Y 277.305,Z 244.943,A -85,B 0,C 180,E1 -17407.36,E2 -17407.36} C_VEL
LIN {X 0,Y 277.21,Z 244.957,A -85,B 0,C 180,E1 -17411.236,E2 -17411.236} C_VEL
LIN {X 0,Y 277.201,Z 244.953,A -85,B 0,C 180,E1 -17415.226,E2 -17415.226} C_VEL
LIN {X 0,Y 277.223,Z 244.956,A -85,B 0,C 180,E1 -17419.512,E2 -17419.512} C_VEL
LIN {X 0,Y 277.268,Z 244.946,A -85,B 0,C 180,E1 -17422.531,E2 -17422.531} C_VEL
LIN {X 0,Y 277.247,Z 244.948,A -85,B 0,C 180,E1 -17426.104,E2 -17426.104} C_VEL
LIN {X 0,Y 277.261,Z 244.942,A -85,B 0,C 180,E1 -17429.539,E2 -17429.539} C_VEL
LIN {X 0,Y 277.358,Z 244.926,A -85,B 0,C 180,E1 -17432.864,E2 -17432.864} C_VEL
LIN {X 0,Y 277.329,Z 244.934,A -85,B 0,C 180,E1 -17436.08,E2 -17436.08} C_VEL
LIN {X 0,Y 277.345,Z 244.929,A -85,B 0,C 180,E1 -17440.766,E2 -17440.766} C_VEL
LIN {X 0,Y 277.435,Z 244.915,A -85,B 0,C 180,E1 -17445.326,E2 -17445.326} C_VEL
LIN {X 0,Y 277.507,Z 244.909,A -85,B 0,C 180,E1 -17449.789,E2 -17449.789} C_VEL
LIN {X 0,Y 277.649,Z 244.9,A -85,B 0,C 180,E1 -17452.729,E2 -17452.729} C_VEL
LIN {X 0,Y 277.821,Z 244.874,A -85,B 0,C 180,E1 -17458.551,E2 -17458.551} C_VEL
LIN {X 0,Y 277.821,Z 244.878,A -85,B 0,C 180,E1 -17461.45,E2 -17461.45} C_VEL
LIN {X 0,Y 277.653,Z 244.893,A -85,B 0,C 180,E1 -17467.271,E2 -17467.271} C_VEL
LIN {X 0,Y 277.507,Z 244.918,A -85,B 0,C 180,E1 -17470.211,E2 -17470.211} C_VEL
LIN {X 0,Y 277.435,Z 244.922,A -85,B 0,C 180,E1 -17474.674,E2 -17474.674} C_VEL
LIN {X 0,Y 277.345,Z 244.937,A -85,B 0,C 180,E1 -17479.234,E2 -17479.234} C_VEL
LIN {X 0,Y 277.287,Z 244.942,A -85,B 0,C 180,E1 -17483.925,E2 -17483.925} C_VEL
LIN {X 0,Y 277.281,Z 244.947,A -85,B 0,C 180,E1 -17487.487,E2 -17487.487} C_VEL
LIN {X 0,Y 277.291,Z 245.049,A -85,B 0,C 180,E1 -17491.922,E2 -17491.922} C_VEL
LIN {X 0,Y 278.655,Z 250.092,A -85,B 0,C 180,E1 -17493.941,E2 -17493.941} C_VEL
LIN {X 0,Y 286.928,Z 266.28,A -85,B 0,C 180,E1 -17495.601,E2 -17495.601} C_VEL
LIN {X 0,Y 293.302,Z 280.946,A -85,B 0,C 180,E1 -17496.854,E2 -17496.854} C_VEL
LIN {X 0,Y 294.916,Z 285.494,A -85,B 0,C 180,E1 -17497.181,E2 -17497.181} C_VEL
LIN {X 0,Y 295.039,Z 288.41,A -85,B 0,C 180,E1 -17497.281,E2 -17497.281} C_VEL
LIN {X 0,Y 292.46,Z 357.437,A -85,B 0,C 180,E1 -17499.044,E2 -17499.044} C_VEL
LIN {X 0,Y 291.498,Z 370.589,A -85,B 0,C 180,E1 -17499.642,E2 -17499.642} C_VEL
LIN {X 0,Y 290.161,Z 383.409,A -85,B 0,C 180,E1 -17500.508,E2 -17500.508} C_VEL
LIN {X 0,Y 288.737,Z 394.572,A -85,B 0,C 180,E1 -17501.542,E2 -17501.542} C_VEL
LIN {X 0,Y 286.799,Z 406.379,A -85,B 0,C 180,E1 -17502.952,E2 -17502.952} C_VEL
LIN {X 0,Y 284.803,Z 416.974,A -85,B 0,C 180,E1 -17504.558,E2 -17504.558} C_VEL
LIN {X 0,Y 282.762,Z 426.673,A -85,B 0,C 180,E1 -17506.42,E2 -17506.42} C_VEL
LIN {X 0,Y 281.069,Z 434.289,A -85,B 0,C 180,E1 -17508.228,E2 -17508.228} C_VEL
LIN {X 0,Y 279.265,Z 442.133,A -85,B 0,C 180,E1 -17510.547,E2 -17510.547} C_VEL
LIN {X 0,Y 277.995,Z 447.721,A -85,B 0,C 180,E1 -17512.646,E2 -17512.646} C_VEL
LIN {X 0,Y 276.811,Z 452.881,A -85,B 0,C 180,E1 -17515.162,E2 -17515.162} C_VEL
LIN {X 0,Y 276.014,Z 456.59,A -85,B 0,C 180,E1 -17517.676,E2 -17517.676} C_VEL
LIN {X 0,Y 275.382,Z 459.032,A -85,B 0,C 180,E1 -17520.194,E2 -17520.194} C_VEL
LIN {X 0,Y 275.011,Z 460.395,A -85,B 0,C 180,E1 -17523.437,E2 -17523.437} C_VEL
LIN {X 0,Y 274.909,Z 460.143,A -85,B 0,C 180,E1 -17525.856,E2 -17525.856} C_VEL
LIN {X 0,Y 275,Z 459.387,A -85,B 0,C 180,E1 -17527.459,E2 -17527.459} C_VEL
LIN {X 0,Y 275.177,Z 458.147,A -85,B 0,C 180,E1 -17529.05,E2 -17529.05} C_VEL
LIN {X 0,Y 275.673,Z 455.309,A -85,B 0,C 180,E1 -17531.458,E2 -17531.458} C_VEL
LIN {X 0,Y 276.201,Z 451.487,A -85,B 0,C 180,E1 -17533.746,E2 -17533.746} C_VEL
LIN {X 0,Y 276.969,Z 446.385,A -85,B 0,C 180,E1 -17536.051,E2 -17536.051} C_VEL
LIN {X 0,Y 278.055,Z 439.906,A -85,B 0,C 180,E1 -17538.334,E2 -17538.334} C_VEL
LIN {X 0,Y 279.198,Z 433.25,A -85,B 0,C 180,E1 -17540.217,E2 -17540.217} C_VEL
LIN {X 0,Y 280.578,Z 425.213,A -85,B 0,C 180,E1 -17542.081,E2 -17542.081} C_VEL
LIN {X 0,Y 282.162,Z 415.336,A -85,B 0,C 180,E1 -17543.923,E2 -17543.923} C_VEL
LIN {X 0,Y 283.644,Z 405.632,A -85,B 0,C 180,E1 -17545.381,E2 -17545.381} C_VEL
LIN {X 0,Y 285.041,Z 395.224,A -85,B 0,C 180,E1 -17546.643,E2 -17546.643} C_VEL
LIN {X 0,Y 286.316,Z 384.016,A -85,B 0,C 180,E1 -17547.714,E2 -17547.714} C_VEL
LIN {X 0,Y 287.364,Z 371.206,A -85,B 0,C 180,E1 -17548.628,E2 -17548.628} C_VEL
LIN {X 0,Y 288.209,Z 357.611,A -85,B 0,C 180,E1 -17549.273,E2 -17549.273} C_VEL
LIN {X 0,Y 290.086,Z 298.682,A -85,B 0,C 180,E1 -17550.791,E2 -17550.791} C_VEL
LIN {X 0,Y 290.435,Z 283.777,A -85,B 0,C 180,E1 -17551.175,E2 -17551.175} C_VEL
LIN {X 0,Y 288.782,Z 275.946,A -85,B 0,C 180,E1 -17551.536,E2 -17551.536} C_VEL
LIN {X 0,Y 281.053,Z 255.337,A -85,B 0,C 180,E1 -17552.825,E2 -17552.825} C_VEL
LIN {X 0,Y 278.514,Z 249.379,A -85,B 0,C 180,E1 -17553.255,E2 -17553.255} C_VEL
LIN {X 0,Y 277.486,Z 244.924,A -85,B 0,C 180,E1 -17554.994,E2 -17554.994} C_VEL
LIN {X 0,Y 277.603,Z 244.907,A -85,B 0,C 180,E1 -17557.272,E2 -17557.272} C_VEL
LIN {X 0,Y 277.46,Z 244.923,A -85,B 0,C 180,E1 -17560.213,E2 -17560.213} C_VEL
LIN {X 0,Y 277.437,Z 244.927,A -85,B 0,C 180,E1 -17564.674,E2 -17564.674} C_VEL
LIN {X 0,Y 277.346,Z 244.938,A -85,B 0,C 180,E1 -17569.233,E2 -17569.233} C_VEL
LIN {X 0,Y 277.288,Z 244.943,A -85,B 0,C 180,E1 -17573.924,E2 -17573.924} C_VEL
LIN {X 0,Y 277.275,Z 244.945,A -85,B 0,C 180,E1 -17577.484,E2 -17577.484} C_VEL
LIN {X 0,Y 277.248,Z 244.948,A -85,B 0,C 180,E1 -17580.472,E2 -17580.472} C_VEL
LIN {X 0,Y 277.247,Z 244.948,A -85,B 0,C 180,E1 -17583.895,E2 -17583.895} C_VEL
LIN {X 0,Y 277.272,Z 244.943,A -85,B 0,C 180,E1 -17587.468,E2 -17587.468} C_VEL
LIN {X 0,Y 277.209,Z 244.952,A -85,B 0,C 180,E1 -17591.236,E2 -17591.236} C_VEL
LIN {X 0,Y 277.2,Z 244.947,A -85,B 0,C 180,E1 -17595.226,E2 -17595.226} C_VEL
LIN {X 0,Y 277.222,Z 244.952,A -85,B 0,C 180,E1 -17599.512,E2 -17599.512} C_VEL
LIN {X 0,Y 277.271,Z 244.938,A -85,B 0,C 180,E1 -17602.531,E2 -17602.531} C_VEL
LIN {X 0,Y 277.246,Z 244.944,A -85,B 0,C 180,E1 -17606.104,E2 -17606.104} C_VEL
LIN {X 0,Y 277.26,Z 244.946,A -85,B 0,C 180,E1 -17609.538,E2 -17609.538} C_VEL
LIN {X 0,Y 277.356,Z 244.93,A -85,B 0,C 180,E1 -17612.864,E2 -17612.864} C_VEL
LIN {X 0,Y 277.327,Z 244.927,A -85,B 0,C 180,E1 -17616.079,E2 -17616.079} C_VEL
LIN {X 0,Y 277.343,Z 244.935,A -85,B 0,C 180,E1 -17620.766,E2 -17620.766} C_VEL
LIN {X 0,Y 277.433,Z 244.921,A -85,B 0,C 180,E1 -17625.326,E2 -17625.326} C_VEL
LIN {X 0,Y 277.413,Z 244.921,A -85,B 0,C 180,E1 -17625.65,E2 -17625.65} C_VEL
LIN {X 0,Y 276.724,Z 245.005,A -85,B 0,C 180,E1 -17626.862,E2 -17626.862} C_VEL
LIN {X 0,Y 273.926,Z 245.345,A -85,B 0,C 180,E1 -17628.84,E2 -17628.84} C_VEL
LIN {X 0,Y 271.6,Z 245.643,A -85,B 0,C 180,E1 -17630.447,E2 -17630.447} C_VEL
LIN {X 0,Y 270.64,Z 245.764,A -85,B 0,C 180,E1 -17631.69,E2 -17631.69} C_VEL
LIN {X 0,Y 270.58,Z 245.773,A -85,B 0,C 180,E1 -17632.111,E2 -17632.111} C_VEL
LIN {X 0,Y 270.629,Z 245.771,A -85,B 0,C 180,E1 -17637.023,E2 -17637.023} C_VEL
LIN {X 0,Y 270.839,Z 245.74,A -85,B 0,C 180,E1 -17640,E2 -17640} C_VEL
LIN {X 0,Y 270.629,Z 245.762,A -85,B 0,C 180,E1 -17642.977,E2 -17642.977} C_VEL
LIN {X 0,Y 270.609,Z 245.774,A -85,B 0,C 180,E1 -17647.461,E2 -17647.461} C_VEL
LIN {X 0,Y 270.44,Z 245.793,A -85,B 0,C 180,E1 -17650.481,E2 -17650.481} C_VEL
LIN {X 0,Y 270.401,Z 245.795,A -85,B 0,C 180,E1 -17655.065,E2 -17655.065} C_VEL
LIN {X 0,Y 270.3,Z 245.814,A -85,B 0,C 180,E1 -17659.756,E2 -17659.756} C_VEL
LIN {X 0,Y 270.272,Z 245.819,A -85,B 0,C 180,E1 -17664.586,E2 -17664.586} C_VEL
LIN {X 0,Y 270.27,Z 245.817,A -85,B 0,C 180,E1 -17667.909,E2 -17667.909} C_VEL
LIN {X 0,Y 270.183,Z 245.828,A -85,B 0,C 180,E1 -17671.348,E2 -17671.348} C_VEL
LIN {X 0,Y 270.2,Z 245.827,A -85,B 0,C 180,E1 -17674.906,E2 -17674.906} C_VEL
LIN {X 0,Y 270.196,Z 245.829,A -85,B 0,C 180,E1 -17678.711,E2 -17678.711} C_VEL
LIN {X 0,Y 270.17,Z 245.825,A -85,B 0,C 180,E1 -17682.559,E2 -17682.559} C_VEL
LIN {X 0,Y 270.168,Z 245.833,A -85,B 0,C 180,E1 -17686.751,E2 -17686.751} C_VEL
LIN {X 0,Y 270.222,Z 245.821,A -85,B 0,C 180,E1 -17691.283,E2 -17691.283} C_VEL
LIN {X 0,Y 270.252,Z 245.851,A -85,B 0,C 180,E1 -17695.103,E2 -17695.103} C_VEL
LIN {X 0,Y 272.575,Z 256.411,A -85,B 0,C 180,E1 -17698.958,E2 -17698.958} C_VEL
LIN {X 0,Y 274.002,Z 263.196,A -85,B 0,C 180,E1 -17701.331,E2 -17701.331} C_VEL
LIN {X 0,Y 278.425,Z 275.571,A -85,B 0,C 180,E1 -17702.133,E2 -17702.133} C_VEL
LIN {X 0,Y 283.371,Z 308.759,A -85,B 0,C 180,E1 -17703.54,E2 -17703.54} C_VEL
LIN {X 0,Y 281.462,Z 372.408,A -85,B 0,C 180,E1 -17705.228,E2 -17705.228} C_VEL
LIN {X 0,Y 280.439,Z 385.971,A -85,B 0,C 180,E1 -17705.871,E2 -17705.871} C_VEL
LIN {X 0,Y 279.125,Z 398.277,A -85,B 0,C 180,E1 -17706.735,E2 -17706.735} C_VEL
LIN {X 0,Y 277.668,Z 410.143,A -85,B 0,C 180,E1 -17707.883,E2 -17707.883} C_VEL
LIN {X 0,Y 275.995,Z 421.573,A -85,B 0,C 180,E1 -17709.31,E2 -17709.31} C_VEL
LIN {X 0,Y 274.201,Z 431.87,A -85,B 0,C 180,E1 -17710.926,E2 -17710.926} C_VEL
LIN {X 0,Y 272.779,Z 441.49,A -85,B 0,C 180,E1 -17712.847,E2 -17712.847} C_VEL
LIN {X 0,Y 271.248,Z 450.145,A -85,B 0,C 180,E1 -17714.984,E2 -17714.984} C_VEL
LIN {X 0,Y 269.934,Z 457.371,A -85,B 0,C 180,E1 -17717.215,E2 -17717.215} C_VEL
LIN {X 0,Y 269.093,Z 463.125,A -85,B 0,C 180,E1 -17719.466,E2 -17719.466} C_VEL
LIN {X 0,Y 268.541,Z 467.643,A -85,B 0,C 180,E1 -17721.724,E2 -17721.724} C_VEL
LIN {X 0,Y 268.225,Z 471.058,A -85,B 0,C 180,E1 -17723.984,E2 -17723.984} C_VEL
LIN {X 0,Y 268.16,Z 472.749,A -85,B 0,C 180,E1 -17725.491,E2 -17725.491} C_VEL
LIN {X 0,Y 268.167,Z 474.031,A -85,B 0,C 180,E1 -17726.996,E2 -17726.996} C_VEL
LIN {X 0,Y 268.188,Z 474.91,A -85,B 0,C 180,E1 -17728.499,E2 -17728.499} C_VEL
LIN {X 0,Y 268.201,Z 475.348,A -85,B 0,C 180,E1 -17730,E2 -17730} C_VEL
LIN {X 0,Y 268.181,Z 475.377,A -85,B 0,C 180,E1 -17731.502,E2 -17731.502} C_VEL
LIN {X 0,Y 268.155,Z 475.016,A -85,B 0,C 180,E1 -17733.005,E2 -17733.005} C_VEL
LIN {X 0,Y 268.163,Z 473.769,A -85,B 0,C 180,E1 -17735.188,E2 -17735.188} C_VEL
LIN {X 0,Y 268.575,Z 470.55,A -85,B 0,C 180,E1 -17738.275,E2 -17738.275} C_VEL
LIN {X 0,Y 269.21,Z 467.005,A -85,B 0,C 180,E1 -17740.53,E2 -17740.53} C_VEL
LIN {X 0,Y 270.115,Z 462.374,A -85,B 0,C 180,E1 -17742.777,E2 -17742.777} C_VEL
LIN {X 0,Y 271.795,Z 455.396,A -85,B 0,C 180,E1 -17745.37,E2 -17745.37} C_VEL
LIN {X 0,Y 273.509,Z 447.869,A -85,B 0,C 180,E1 -17747.573,E2 -17747.573} C_VEL
LIN {X 0,Y 275.19,Z 440.21,A -85,B 0,C 180,E1 -17749.39,E2 -17749.39} C_VEL
LIN {X 0,Y 277.224,Z 430.934,A -85,B 0,C 180,E1 -17751.177,E2 -17751.177} C_VEL
LIN {X 0,Y 279.413,Z 420.633,A -85,B 0,C 180,E1 -17752.751,E2 -17752.751} C_VEL
LIN {X 0,Y 281.46,Z 409.254,A -85,B 0,C 180,E1 -17754.135,E2 -17754.135} C_VEL
LIN {X 0,Y 283.32,Z 397.433,A -85,B 0,C 180,E1 -17755.236,E2 -17755.236} C_VEL
LIN {X 0,Y 284.852,Z 384.442,A -85,B 0,C 180,E1 -17756.12,E2 -17756.12} C_VEL
LIN {X 0,Y 286.02,Z 370.762,A -85,B 0,C 180,E1 -17756.737,E2 -17756.737} C_VEL
LIN {X 0,Y 288.187,Z 309.952,A -85,B 0,C 180,E1 -17758.341,E2 -17758.341} C_VEL
LIN {X 0,Y 285.347,Z 291.046,A -85,B 0,C 180,E1 -17759.281,E2 -17759.281} C_VEL
LIN {X 0,Y 283.634,Z 282.659,A -85,B 0,C 180,E1 -17759.768,E2 -17759.768} C_VEL
LIN {X 0,Y 278.235,Z 270.148,A -85,B 0,C 180,E1 -17760.909,E2 -17760.909} C_VEL
LIN {X 0,Y 274.229,Z 261.812,A -85,B 0,C 180,E1 -17761.789,E2 -17761.789} C_VEL
LIN {X 0,Y 272.279,Z 253.41,A -85,B 0,C 180,E1 -17765.051,E2 -17765.051} C_VEL
LIN {X 0,Y 270.229,Z 245.822,A -85,B 0,C 180,E1 -17768.265,E2 -17768.265} C_VEL
LIN {X 0,Y 270.172,Z 245.828,A -85,B 0,C 180,E1 -17772.558,E2 -17772.558} C_VEL
LIN {X 0,Y 270.165,Z 245.836,A -85,B 0,C 180,E1 -17776.751,E2 -17776.751} C_VEL
LIN {X 0,Y 270.174,Z 245.833,A -85,B 0,C 180,E1 -17779.434,E2 -17779.434} C_VEL
LIN {X 0,Y 270.226,Z 245.822,A -85,B 0,C 180,E1 -17783.73,E2 -17783.73} C_VEL
LIN {X 0,Y 270.203,Z 245.828,A -85,B 0,C 180,E1 -17786.892,E2 -17786.892} C_VEL
LIN {X 0,Y 270.228,Z 245.823,A -85,B 0,C 180,E1 -17790.387,E2 -17790.387} C_VEL
LIN {X 0,Y 270.263,Z 245.816,A -85,B 0,C 180,E1 -17793.764,E2 -17793.764} C_VEL
LIN {X 0,Y 270.233,Z 245.814,A -85,B 0,C 180,E1 -17797.039,E2 -17797.039} C_VEL
LIN {X 0,Y 270.302,Z 245.812,A -85,B 0,C 180,E1 -17800.245,E2 -17800.245} C_VEL
LIN {X 0,Y 270.403,Z 245.794,A -85,B 0,C 180,E1 -17804.935,E2 -17804.935} C_VEL
LIN {X 0,Y 270.442,Z 245.79,A -85,B 0,C 180,E1 -17809.519,E2 -17809.519} C_VEL
LIN {X 0,Y 270.608,Z 245.776,A -85,B 0,C 180,E1 -17812.539,E2 -17812.539} C_VEL
LIN {X 0,Y 270.787,Z 245.75,A -85,B 0,C 180,E1 -17818.513,E2 -17818.513} C_VEL
LIN {X 0,Y 270.787,Z 245.755,A -85,B 0,C 180,E1 -17821.487,E2 -17821.487} C_VEL
LIN {X 0,Y 270.611,Z 245.769,A -85,B 0,C 180,E1 -17827.461,E2 -17827.461} C_VEL
LIN {X 0,Y 270.442,Z 245.797,A -85,B 0,C 180,E1 -17830.481,E2 -17830.481} C_VEL
LIN {X 0,Y 270.403,Z 245.796,A -85,B 0,C 180,E1 -17835.065,E2 -17835.065} C_VEL
LIN {X 0,Y 270.302,Z 245.816,A -85,B 0,C 180,E1 -17839.756,E2 -17839.756} C_VEL
LIN {X 0,Y 270.228,Z 245.825,A -85,B 0,C 180,E1 -17844.59,E2 -17844.59} C_VEL
LIN {X 0,Y 270.209,Z 245.822,A -85,B 0,C 180,E1 -17847.916,E2 -17847.916} C_VEL
LIN {X 0,Y 270.235,Z 246.009,A -85,B 0,C 180,E1 -17851.034,E2 -17851.034} C_VEL
LIN {X 0,Y 271.375,Z 250.188,A -85,B 0,C 180,E1 -17852.836,E2 -17852.836} C_VEL
LIN {X 0,Y 278.547,Z 263.712,A -85,B 0,C 180,E1 -17854.371,E2 -17854.371} C_VEL
LIN {X 0,Y 285.303,Z 278.089,A -85,B 0,C 180,E1 -17855.753,E2 -17855.753} C_VEL
LIN {X 0,Y 288.952,Z 287.307,A -85,B 0,C 180,E1 -17856.508,E2 -17856.508} C_VEL
LIN {X 0,Y 286.273,Z 357.981,A -85,B 0,C 180,E1 -17858.366,E2 -17858.366} C_VEL
LIN {X 0,Y 285.266,Z 371.321,A -85,B 0,C 180,E1 -17858.994,E2 -17858.994} C_VEL
LIN {X 0,Y 283.861,Z 383.93,A -85,B 0,C 180,E1 -17859.869,E2 -17859.869} C_VEL
LIN {X 0,Y 282.094,Z 396.584,A -85,B 0,C 180,E1 -17861.094,E2 -17861.094} C_VEL
LIN {X 0,Y 280.175,Z 407.765,A -85,B 0,C 180,E1 -17862.495,E2 -17862.495} C_VEL
LIN {X 0,Y 278.055,Z 418.328,A -85,B 0,C 180,E1 -17864.177,E2 -17864.177} C_VEL
LIN {X 0,Y 275.922,Z 427.914,A -85,B 0,C 180,E1 -17866.103,E2 -17866.103} C_VEL
LIN {X 0,Y 273.99,Z 436.155,A -85,B 0,C 180,E1 -17868.171,E2 -17868.171} C_VEL
LIN {X 0,Y 272.25,Z 443.256,A -85,B 0,C 180,E1 -17870.415,E2 -17870.415} C_VEL
LIN {X 0,Y 270.989,Z 448.397,A -85,B 0,C 180,E1 -17872.449,E2 -17872.449} C_VEL
LIN {X 0,Y 269.758,Z 453.413,A -85,B 0,C 180,E1 -17875.029,E2 -17875.029} C_VEL
LIN {X 0,Y 269.166,Z 455.988,A -85,B 0,C 180,E1 -17876.748,E2 -17876.748} C_VEL
LIN {X 0,Y 268.668,Z 457.935,A -85,B 0,C 180,E1 -17878.455,E2 -17878.455} C_VEL
LIN {X 0,Y 268.294,Z 459.35,A -85,B 0,C 180,E1 -17880.152,E2 -17880.152} C_VEL
LIN {X 0,Y 267.958,Z 460.572,A -85,B 0,C 180,E1 -17883.095,E2 -17883.095} C_VEL
LIN {X 0,Y 267.819,Z 460.528,A -85,B 0,C 180,E1 -17885.174,E2 -17885.174} C_VEL
LIN {X 0,Y 267.867,Z 459.925,A -85,B 0,C 180,E1 -17886.824,E2 -17886.824} C_VEL
LIN {X 0,Y 267.988,Z 458.862,A -85,B 0,C 180,E1 -17888.46,E2 -17888.46} C_VEL
LIN {X 0,Y 268.346,Z 456.806,A -85,B 0,C 180,E1 -17890.536,E2 -17890.536} C_VEL
LIN {X 0,Y 268.981,Z 452.783,A -85,B 0,C 180,E1 -17893.297,E2 -17893.297} C_VEL
LIN {X 0,Y 269.728,Z 448.014,A -85,B 0,C 180,E1 -17895.668,E2 -17895.668} C_VEL
LIN {X 0,Y 270.769,Z 441.879,A -85,B 0,C 180,E1 -17898.015,E2 -17898.015} C_VEL
LIN {X 0,Y 272.129,Z 434.173,A -85,B 0,C 180,E1 -17900.336,E2 -17900.336} C_VEL
LIN {X 0,Y 273.554,Z 426.275,A -85,B 0,C 180,E1 -17902.248,E2 -17902.248} C_VEL
LIN {X 0,Y 275.168,Z 416.664,A -85,B 0,C 180,E1 -17904.136,E2 -17904.136} C_VEL
LIN {X 0,Y 276.874,Z 405.853,A -85,B 0,C 180,E1 -17905.815,E2 -17905.815} C_VEL
LIN {X 0,Y 278.324,Z 395.447,A -85,B 0,C 180,E1 -17907.105,E2 -17907.105} C_VEL
LIN {X 0,Y 279.794,Z 383.162,A -85,B 0,C 180,E1 -17908.291,E2 -17908.291} C_VEL
LIN {X 0,Y 280.856,Z 369.866,A -85,B 0,C 180,E1 -17909.226,E2 -17909.226} C_VEL
LIN {X 0,Y 281.656,Z 356.942,A -85,B 0,C 180,E1 -17909.83,E2 -17909.83} C_VEL
LIN {X 0,Y 283.954,Z 285.04,A -85,B 0,C 180,E1 -17911.706,E2 -17911.706} C_VEL
LIN {X 0,Y 282.389,Z 277.904,A -85,B 0,C 180,E1 -17912.052,E2 -17912.052} C_VEL
LIN {X 0,Y 275.131,Z 258.505,A -85,B 0,C 180,E1 -17913.305,E2 -17913.305} C_VEL
LIN {X 0,Y 271.217,Z 249.53,A -85,B 0,C 180,E1 -17913.998,E2 -17913.998} C_VEL
LIN {X 0,Y 270.462,Z 245.8,A -85,B 0,C 180,E1 -17915.498,E2 -17915.498} C_VEL
LIN {X 0,Y 270.53,Z 245.788,A -85,B 0,C 180,E1 -17918.967,E2 -17918.967} C_VEL
LIN {X 0,Y 270.361,Z 245.81,A -85,B 0,C 180,E1 -17923.53,E2 -17923.53} C_VEL
LIN {X 0,Y 270.357,Z 245.81,A -85,B 0,C 180,E1 -17926.615,E2 -17926.615} C_VEL
LIN {X 0,Y 270.293,Z 245.815,A -85,B 0,C 180,E1 -17930.6,E2 -17930.6} C_VEL
LIN {X 0,Y 270.231,Z 245.822,A -85,B 0,C 180,E1 -17934.589,E2 -17934.589} C_VEL
LIN {X 0,Y 270.204,Z 245.823,A -85,B 0,C 180,E1 -17937.916,E2 -17937.916} C_VEL
LIN {X 0,Y 270.174,Z 245.83,A -85,B 0,C 180,E1 -17941.349,E2 -17941.349} C_VEL
LIN {X 0,Y 270.202,Z 245.82,A -85,B 0,C 180,E1 -17944.905,E2 -17944.905} C_VEL
LIN {X 0,Y 270.198,Z 245.826,A -85,B 0,C 180,E1 -17948.71,E2 -17948.71} C_VEL
LIN {X 0,Y 270.171,Z 245.824,A -85,B 0,C 180,E1 -17952.558,E2 -17952.558} C_VEL
LIN {X 0,Y 270.165,Z 245.828,A -85,B 0,C 180,E1 -17956.75,E2 -17956.75} C_VEL
LIN {X 0,Y 270.173,Z 245.83,A -85,B 0,C 180,E1 -17959.434,E2 -17959.434} C_VEL
LIN {X 0,Y 270.226,Z 245.814,A -85,B 0,C 180,E1 -17963.73,E2 -17963.73} C_VEL
LIN {X 0,Y 270.201,Z 245.821,A -85,B 0,C 180,E1 -17966.892,E2 -17966.892} C_VEL
LIN {X 0,Y 270.194,Z 245.827,A -85,B 0,C 180,E1 -17970.382,E2 -17970.382} C_VEL
LIN {X 0,Y 270.262,Z 245.814,A -85,B 0,C 180,E1 -17973.763,E2 -17973.763} C_VEL
LIN {X 0,Y 270.231,Z 245.809,A -85,B 0,C 180,E1 -17977.038,E2 -17977.038} C_VEL
LIN {X 0,Y 270.3,Z 245.815,A -85,B 0,C 180,E1 -17980.244,E2 -17980.244} C_VEL
LIN {X 0,Y 270.401,Z 245.797,A -85,B 0,C 180,E1 -17984.935,E2 -17984.935} C_VEL
LIN {X 0,Y 270.44,Z 245.779,A -85,B 0,C 180,E1 -17989.519,E2 -17989.519} C_VEL
LIN {X 0,Y 270.58,Z 245.773,A -85,B 0,C 180,E1 -17992.111,E2 -17992.111} C_VEL
LIN {X 0,Y 269.981,Z 245.856,A -85,B 0,C 180,E1 -17993.351,E2 -17993.351} C_VEL
LIN {X 0,Y 267.222,Z 246.206,A -85,B 0,C 180,E1 -17995.374,E2 -17995.374} C_VEL
LIN {X 0,Y 264.849,Z 246.497,A -85,B 0,C 180,E1 -17997.018,E2 -17997.018} C_VEL
LIN {X 0,Y 263.828,Z 246.617,A -85,B 0,C 180,E1 -17998.292,E2 -17998.292} C_VEL
LIN {X 0,Y 263.745,Z 246.624,A -85,B 0,C 180,E1 -17998.723,E2 -17998.723} C_VEL
LIN {X 0,Y 263.749,Z 246.615,A -85,B 0,C 180,E1 -18001.527,E2 -18001.527} C_VEL
LIN {X 0,Y 263.571,Z 246.652,A -85,B 0,C 180,E1 -18007.662,E2 -18007.662} C_VEL
LIN {X 0,Y 263.372,Z 246.672,A -85,B 0,C 180,E1 -18010.766,E2 -18010.766} C_VEL
LIN {X 0,Y 263.349,Z 246.673,A -85,B 0,C 180,E1 -18015.478,E2 -18015.478} C_VEL
LIN {X 0,Y 263.262,Z 246.691,A -85,B 0,C 180,E1 -18020.307,E2 -18020.307} C_VEL
LIN {X 0,Y 263.207,Z 246.697,A -85,B 0,C 180,E1 -18025.291,E2 -18025.291} C_VEL
LIN {X 0,Y 263.178,Z 246.699,A -85,B 0,C 180,E1 -18028.73,E2 -18028.73} C_VEL
LIN {X 0,Y 263.131,Z 246.709,A -85,B 0,C 180,E1 -18032.288,E2 -18032.288} C_VEL
LIN {X 0,Y 263.181,Z 246.7,A -85,B 0,C 180,E1 -18036.764,E2 -18036.764} C_VEL
LIN {X 0,Y 263.123,Z 246.705,A -85,B 0,C 180,E1 -18041.594,E2 -18041.594} C_VEL
LIN {X 0,Y 263.124,Z 246.712,A -85,B 0,C 180,E1 -18046.151,E2 -18046.151} C_VEL
LIN {X 0,Y 263.121,Z 246.711,A -85,B 0,C 180,E1 -18050.131,E2 -18050.131} C_VEL
LIN {X 0,Y 263.256,Z 246.83,A -85,B 0,C 180,E1 -18054.598,E2 -18054.598} C_VEL
LIN {X 0,Y 265.371,Z 256.534,A -85,B 0,C 180,E1 -18058.256,E2 -18058.256} C_VEL
LIN {X 0,Y 266.746,Z 263.069,A -85,B 0,C 180,E1 -18060.606,E2 -18060.606} C_VEL
LIN {X 0,Y 272.139,Z 277.933,A -85,B 0,C 180,E1 -18061.603,E2 -18061.603} C_VEL
LIN {X 0,Y 276.717,Z 308.461,A -85,B 0,C 180,E1 -18062.937,E2 -18062.937} C_VEL
LIN {X 0,Y 276.605,Z 319.064,A -85,B 0,C 180,E1 -18063.236,E2 -18063.236} C_VEL
LIN {X 0,Y 274.939,Z 371.428,A -85,B 0,C 180,E1 -18064.649,E2 -18064.649} C_VEL
LIN {X 0,Y 273.864,Z 385.238,A -85,B 0,C 180,E1 -18065.304,E2 -18065.304} C_VEL
LIN {X 0,Y 272.467,Z 398.234,A -85,B 0,C 180,E1 -18066.233,E2 -18066.233} C_VEL
LIN {X 0,Y 270.839,Z 410.858,A -85,B 0,C 180,E1 -18067.496,E2 -18067.496} C_VEL
LIN {X 0,Y 269.118,Z 422.123,A -85,B 0,C 180,E1 -18068.957,E2 -18068.957} C_VEL
LIN {X 0,Y 267.273,Z 432.245,A -85,B 0,C 180,E1 -18070.612,E2 -18070.612} C_VEL
LIN {X 0,Y 265.882,Z 441.358,A -85,B 0,C 180,E1 -18072.487,E2 -18072.487} C_VEL
LIN {X 0,Y 264.337,Z 449.659,A -85,B 0,C 180,E1 -18074.582,E2 -18074.582} C_VEL
LIN {X 0,Y 262.957,Z 456.944,A -85,B 0,C 180,E1 -18076.869,E2 -18076.869} C_VEL
LIN {X 0,Y 262.069,Z 462.756,A -85,B 0,C 180,E1 -18079.18,E2 -18079.18} C_VEL
LIN {X 0,Y 261.503,Z 467.317,A -85,B 0,C 180,E1 -18081.5,E2 -18081.5} C_VEL
LIN {X 0,Y 261.153,Z 470.768,A -85,B 0,C 180,E1 -18083.821,E2 -18083.821} C_VEL
LIN {X 0,Y 261.067,Z 472.477,A -85,B 0,C 180,E1 -18085.368,E2 -18085.368} C_VEL
LIN {X 0,Y 261.082,Z 473.776,A -85,B 0,C 180,E1 -18086.914,E2 -18086.914} C_VEL
LIN {X 0,Y 261.116,Z 474.673,A -85,B 0,C 180,E1 -18088.458,E2 -18088.458} C_VEL
LIN {X 0,Y 261.126,Z 475.143,A -85,B 0,C 180,E1 -18090,E2 -18090} C_VEL
LIN {X 0,Y 261.108,Z 475.188,A -85,B 0,C 180,E1 -18091.543,E2 -18091.543} C_VEL
LIN {X 0,Y 261.05,Z 474.842,A -85,B 0,C 180,E1 -18093.087,E2 -18093.087} C_VEL
LIN {X 0,Y 261.085,Z 473.772,A -85,B 0,C 180,E1 -18095.137,E2 -18095.137} C_VEL
LIN {X 0,Y 261.361,Z 471.379,A -85,B 0,C 180,E1 -18097.727,E2 -18097.727} C_VEL
LIN {X 0,Y 261.948,Z 468.218,A -85,B 0,C 180,E1 -18100.044,E2 -18100.044} C_VEL
LIN {X 0,Y 262.803,Z 464.005,A -85,B 0,C 180,E1 -18102.353,E2 -18102.353} C_VEL
LIN {X 0,Y 264.4,Z 457.611,A -85,B 0,C 180,E1 -18105.021,E2 -18105.021} C_VEL
LIN {X 0,Y 266.179,Z 450.67,A -85,B 0,C 180,E1 -18107.28,E2 -18107.28} C_VEL
LIN {X 0,Y 267.909,Z 443.062,A -85,B 0,C 180,E1 -18109.282,E2 -18109.282} C_VEL
LIN {X 0,Y 270.195,Z 433.151,A -85,B 0,C 180,E1 -18111.355,E2 -18111.355} C_VEL
LIN {X 0,Y 272.636,Z 422.274,A -85,B 0,C 180,E1 -18113.148,E2 -18113.148} C_VEL
LIN {X 0,Y 274.753,Z 411.339,A -85,B 0,C 180,E1 -18114.561,E2 -18114.561} C_VEL
LIN {X 0,Y 276.806,Z 399.155,A -85,B 0,C 180,E1 -18115.772,E2 -18115.772} C_VEL
LIN {X 0,Y 278.491,Z 386.41,A -85,B 0,C 180,E1 -18116.713,E2 -18116.713} C_VEL
LIN {X 0,Y 279.724,Z 373.226,A -85,B 0,C 180,E1 -18117.366,E2 -18117.366} C_VEL
LIN {X 0,Y 280.701,Z 351.376,A -85,B 0,C 180,E1 -18118.002,E2 -18118.002} C_VEL
LIN {X 0,Y 282.145,Z 310.61,A -85,B 0,C 180,E1 -18119.087,E2 -18119.087} C_VEL
LIN {X 0,Y 278.879,Z 289.588,A -85,B 0,C 180,E1 -18120.192,E2 -18120.192} C_VEL
LIN {X 0,Y 277.805,Z 284.899,A -85,B 0,C 180,E1 -18120.491,E2 -18120.491} C_VEL
LIN {X 0,Y 272.596,Z 273.125,A -85,B 0,C 180,E1 -18121.639,E2 -18121.639} C_VEL
LIN {X 0,Y 267.017,Z 261.574,A -85,B 0,C 180,E1 -18122.918,E2 -18122.918} C_VEL
LIN {X 0,Y 265.074,Z 253.594,A -85,B 0,C 180,E1 -18126.182,E2 -18126.182} C_VEL
LIN {X 0,Y 263.131,Z 246.708,A -85,B 0,C 180,E1 -18129.295,E2 -18129.295} C_VEL
LIN {X 0,Y 263.124,Z 246.707,A -85,B 0,C 180,E1 -18131.893,E2 -18131.893} C_VEL
LIN {X 0,Y 263.124,Z 246.711,A -85,B 0,C 180,E1 -18136.151,E2 -18136.151} C_VEL
LIN {X 0,Y 263.106,Z 246.712,A -85,B 0,C 180,E1 -18140.128,E2 -18140.128} C_VEL
LIN {X 0,Y 263.163,Z 246.7,A -85,B 0,C 180,E1 -18144.018,E2 -18144.018} C_VEL
LIN {X 0,Y 263.133,Z 246.702,A -85,B 0,C 180,E1 -18147.712,E2 -18147.712} C_VEL
LIN {X 0,Y 263.201,Z 246.693,A -85,B 0,C 180,E1 -18151.783,E2 -18151.783} C_VEL
LIN {X 0,Y 263.226,Z 246.696,A -85,B 0,C 180,E1 -18155.2,E2 -18155.2} C_VEL
LIN {X 0,Y 263.264,Z 246.69,A -85,B 0,C 180,E1 -18159.693,E2 -18159.693} C_VEL
LIN {X 0,Y 263.351,Z 246.677,A -85,B 0,C 180,E1 -18164.522,E2 -18164.522} C_VEL
LIN {X 0,Y 263.374,Z 246.672,A -85,B 0,C 180,E1 -18169.234,E2 -18169.234} C_VEL
LIN {X 0,Y 263.57,Z 246.651,A -85,B 0,C 180,E1 -18172.338,E2 -18172.338} C_VEL
LIN {X 0,Y 263.751,Z 246.626,A -85,B 0,C 180,E1 -18178.473,E2 -18178.473} C_VEL
LIN {X 0,Y 263.751,Z 246.631,A -85,B 0,C 180,E1 -18181.527,E2 -18181.527} C_VEL
LIN {X 0,Y 263.573,Z 246.645,A -85,B 0,C 180,E1 -18187.662,E2 -18187.662} C_VEL
LIN {X 0,Y 263.374,Z 246.674,A -85,B 0,C 180,E1 -18190.766,E2 -18190.766} C_VEL
LIN {X 0,Y 263.351,Z 246.675,A -85,B 0,C 180,E1 -18195.478,E2 -18195.478} C_VEL
LIN {X 0,Y 263.263,Z 246.692,A -85,B 0,C 180,E1 -18200.307,E2 -18200.307} C_VEL
LIN {X 0,Y 263.173,Z 246.705,A -85,B 0,C 180,E1 -18205.295,E2 -18205.295} C_VEL
LIN {X 0,Y 263.138,Z 246.699,A -85,B 0,C 180,E1 -18209.831,E2 -18209.831} C_VEL
LIN {X 0,Y 263.171,Z 246.881,A -85,B 0,C 180,E1 -18210.048,E2 -18210.048} C_VEL
LIN {X 0,Y 264.247,Z 250.7,A -85,B 0,C 180,E1 -18211.687,E2 -18211.687} C_VEL
LIN {X 0,Y 271.651,Z 264.099,A -85,B 0,C 180,E1 -18213.354,E2 -18213.354} C_VEL
LIN {X 0,Y 277.968,Z 277.217,A -85,B 0,C 180,E1 -18214.727,E2 -18214.727} C_VEL
LIN {X 0,Y 282.933,Z 289.165,A -85,B 0,C 180,E1 -18215.786,E2 -18215.786} C_VEL
LIN {X 0,Y 280.142,Z 358.467,A -85,B 0,C 180,E1 -18217.645,E2 -18217.645} C_VEL
LIN {X 0,Y 279.044,Z 372.104,A -85,B 0,C 180,E1 -18218.307,E2 -18218.307} C_VEL
LIN {X 0,Y 277.684,Z 383.817,A -85,B 0,C 180,E1 -18219.14,E2 -18219.14} C_VEL
LIN {X 0,Y 276.106,Z 395.002,A -85,B 0,C 180,E1 -18220.216,E2 -18220.216} C_VEL
LIN {X 0,Y 274.001,Z 406.864,A -85,B 0,C 180,E1 -18221.693,E2 -18221.693} C_VEL
LIN {X 0,Y 271.817,Z 417.355,A -85,B 0,C 180,E1 -18223.349,E2 -18223.349} C_VEL
LIN {X 0,Y 269.596,Z 426.949,A -85,B 0,C 180,E1 -18225.263,E2 -18225.263} C_VEL
LIN {X 0,Y 267.543,Z 435.306,A -85,B 0,C 180,E1 -18227.352,E2 -18227.352} C_VEL
LIN {X 0,Y 265.76,Z 442.306,A -85,B 0,C 180,E1 -18229.535,E2 -18229.535} C_VEL
LIN {X 0,Y 264.507,Z 447.058,A -85,B 0,C 180,E1 -18231.362,E2 -18231.362} C_VEL
LIN {X 0,Y 263.104,Z 452.506,A -85,B 0,C 180,E1 -18234.009,E2 -18234.009} C_VEL
LIN {X 0,Y 262.263,Z 455.831,A -85,B 0,C 180,E1 -18236.174,E2 -18236.174} C_VEL
LIN {X 0,Y 261.811,Z 457.47,A -85,B 0,C 180,E1 -18237.529,E2 -18237.529} C_VEL
LIN {X 0,Y 261.342,Z 459.155,A -85,B 0,C 180,E1 -18239.378,E2 -18239.378} C_VEL
LIN {X 0,Y 261.048,Z 460.155,A -85,B 0,C 180,E1 -18241.014,E2 -18241.014} C_VEL
LIN {X 0,Y 260.891,Z 460.749,A -85,B 0,C 180,E1 -18242.745,E2 -18242.745} C_VEL
LIN {X 0,Y 260.738,Z 460.803,A -85,B 0,C 180,E1 -18244.452,E2 -18244.452} C_VEL
LIN {X 0,Y 260.735,Z 460.315,A -85,B 0,C 180,E1 -18246.414,E2 -18246.414} C_VEL
LIN {X 0,Y 260.831,Z 459.531,A -85,B 0,C 180,E1 -18247.838,E2 -18247.838} C_VEL
LIN {X 0,Y 261.224,Z 457.325,A -85,B 0,C 180,E1 -18250.33,E2 -18250.33} C_VEL
LIN {X 0,Y 261.784,Z 453.983,A -85,B 0,C 180,E1 -18252.824,E2 -18252.824} C_VEL
LIN {X 0,Y 262.52,Z 449.234,A -85,B 0,C 180,E1 -18255.393,E2 -18255.393} C_VEL
LIN {X 0,Y 263.679,Z 442.67,A -85,B 0,C 180,E1 -18258.079,E2 -18258.079} C_VEL
LIN {X 0,Y 265.11,Z 434.977,A -85,B 0,C 180,E1 -18260.492,E2 -18260.492} C_VEL
LIN {X 0,Y 266.854,Z 425.622,A -85,B 0,C 180,E1 -18262.813,E2 -18262.813} C_VEL
LIN {X 0,Y 268.508,Z 416.125,A -85,B 0,C 180,E1 -18264.679,E2 -18264.679} C_VEL
LIN {X 0,Y 270.13,Z 406.052,A -85,B 0,C 180,E1 -18266.27,E2 -18266.27} C_VEL
LIN {X 0,Y 271.62,Z 395.65,A -85,B 0,C 180,E1 -18267.59,E2 -18267.59} C_VEL
LIN {X 0,Y 272.97,Z 384.648,A -85,B 0,C 180,E1 -18268.69,E2 -18268.69} C_VEL
LIN {X 0,Y 274.099,Z 372.101,A -85,B 0,C 180,E1 -18269.636,E2 -18269.636} C_VEL
LIN {X 0,Y 275.013,Z 358.66,A -85,B 0,C 180,E1 -18270.313,E2 -18270.313} C_VEL
LIN {X 0,Y 276.069,Z 329.861,A -85,B 0,C 180,E1 -18271.119,E2 -18271.119} C_VEL
LIN {X 0,Y 277.369,Z 285.53,A -85,B 0,C 180,E1 -18272.295,E2 -18272.295} C_VEL
LIN {X 0,Y 276.135,Z 280.19,A -85,B 0,C 180,E1 -18272.567,E2 -18272.567} C_VEL
LIN {X 0,Y 269.121,Z 261.428,A -85,B 0,C 180,E1 -18273.818,E2 -18273.818} C_VEL
LIN {X 0,Y 264.029,Z 249.792,A -85,B 0,C 180,E1 -18274.723,E2 -18274.723} C_VEL
LIN {X 0,Y 263.476,Z 246.672,A -85,B 0,C 180,E1 -18276.029,E2 -18276.029} C_VEL
LIN {X 0,Y 263.491,Z 246.663,A -85,B 0,C 180,E1 -18279.287,E2 -18279.287} C_VEL
LIN {X 0,Y 263.31,Z 246.689,A -85,B 0,C 180,E1 -18283.899,E2 -18283.899} C_VEL
LIN {X 0,Y 263.273,Z 246.693,A -85,B 0,C 180,E1 -18287.076,E2 -18287.076} C_VEL
LIN {X 0,Y 263.216,Z 246.697,A -85,B 0,C 180,E1 -18290.849,E2 -18290.849} C_VEL
LIN {X 0,Y 263.176,Z 246.701,A -85,B 0,C 180,E1 -18295.294,E2 -18295.294} C_VEL
LIN {X 0,Y 263.137,Z 246.7,A -85,B 0,C 180,E1 -18298.734,E2 -18298.734} C_VEL
LIN {X 0,Y 263.129,Z 246.708,A -85,B 0,C 180,E1 -18302.288,E2 -18302.288} C_VEL
LIN {X 0,Y 263.185,Z 246.696,A -85,B 0,C 180,E1 -18306.763,E2 -18306.763} C_VEL
LIN {X 0,Y 263.124,Z 246.708,A -85,B 0,C 180,E1 -18311.593,E2 -18311.593} C_VEL
LIN {X 0,Y 263.124,Z 246.706,A -85,B 0,C 180,E1 -18316.15,E2 -18316.15} C_VEL
LIN {X 0,Y 263.105,Z 246.711,A -85,B 0,C 180,E1 -18320.127,E2 -18320.127} C_VEL
LIN {X 0,Y 263.163,Z 246.691,A -85,B 0,C 180,E1 -18324.018,E2 -18324.018} C_VEL
LIN {X 0,Y 263.131,Z 246.704,A -85,B 0,C 180,E1 -18327.711,E2 -18327.711} C_VEL
LIN {X 0,Y 263.195,Z 246.7,A -85,B 0,C 180,E1 -18331.785,E2 -18331.785} C_VEL
LIN {X 0,Y 263.225,Z 246.682,A -85,B 0,C 180,E1 -18335.2,E2 -18335.2} C_VEL
LIN {X 0,Y 263.262,Z 246.686,A -85,B 0,C 180,E1 -18339.693,E2 -18339.693} C_VEL
LIN {X 0,Y 263.349,Z 246.677,A -85,B 0,C 180,E1 -18344.522,E2 -18344.522} C_VEL
LIN {X 0,Y 263.372,Z 246.657,A -85,B 0,C 180,E1 -18349.234,E2 -18349.234} C_VEL
LIN {X 0,Y 263.571,Z 246.649,A -85,B 0,C 180,E1 -18352.338,E2 -18352.338} C_VEL
LIN {X 0,Y 263.75,Z 246.626,A -85,B 0,C 180,E1 -18358.473,E2 -18358.473} C_VEL
LIN {X 0,Y 263.745,Z 246.624,A -85,B 0,C 180,E1 -18358.723,E2 -18358.723} C_VEL
LIN {X 0,Y 263.406,Z 246.667,A -85,B 0,C 180,E1 -18359.576,E2 -18359.576} C_VEL
LIN {X 0,Y 261.974,Z 246.838,A -85,B 0,C 180,E1 -18360.831,E2 -18360.831} C_VEL
LIN {X 0,Y 257.458,Z 247.404,A -85,B 0,C 180,E1 -18363.754,E2 -18363.754} C_VEL
LIN {X 0,Y 256.436,Z 247.537,A -85,B 0,C 180,E1 -18365.066,E2 -18365.066} C_VEL
LIN {X 0,Y 256.388,Z 247.542,A -85,B 0,C 180,E1 -18365.511,E2 -18365.511} C_VEL
LIN {X 0,Y 256.538,Z 247.529,A -85,B 0,C 180,E1 -18367.873,E2 -18367.873} C_VEL
LIN {X 0,Y 256.308,Z 247.55,A -85,B 0,C 180,E1 -18371.066,E2 -18371.066} C_VEL
LIN {X 0,Y 256.298,Z 247.553,A -85,B 0,C 180,E1 -18375.915,E2 -18375.915} C_VEL
LIN {X 0,Y 256.165,Z 247.571,A -85,B 0,C 180,E1 -18380.895,E2 -18380.895} C_VEL
LIN {X 0,Y 256.187,Z 247.571,A -85,B 0,C 180,E1 -18385.139,E2 -18385.139} C_VEL
LIN {X 0,Y 256.112,Z 247.578,A -85,B 0,C 180,E1 -18389.6,E2 -18389.6} C_VEL
LIN {X 0,Y 256.066,Z 247.583,A -85,B 0,C 180,E1 -18393.293,E2 -18393.293} C_VEL
LIN {X 0,Y 256.113,Z 247.579,A -85,B 0,C 180,E1 -18397.271,E2 -18397.271} C_VEL
LIN {X 0,Y 256.053,Z 247.585,A -85,B 0,C 180,E1 -18401.204,E2 -18401.204} C_VEL
LIN {X 0,Y 256.053,Z 247.59,A -85,B 0,C 180,E1 -18405.531,E2 -18405.531} C_VEL
LIN {X 0,Y 256.062,Z 247.589,A -85,B 0,C 180,E1 -18408.799,E2 -18408.799} C_VEL
LIN {X 0,Y 256.145,Z 247.582,A -85,B 0,C 180,E1 -18412.87,E2 -18412.87} C_VEL
LIN {X 0,Y 256.194,Z 247.581,A -85,B 0,C 180,E1 -18413.98,E2 -18413.98} C_VEL
LIN {X 0,Y 258.604,Z 258.621,A -85,B 0,C 180,E1 -18418.26,E2 -18418.26} C_VEL
LIN {X 0,Y 259.488,Z 262.852,A -85,B 0,C 180,E1 -18419.828,E2 -18419.828} C_VEL
LIN {X 0,Y 265.842,Z 279.824,A -85,B 0,C 180,E1 -18421.033,E2 -18421.033} C_VEL
LIN {X 0,Y 270.337,Z 310.356,A -85,B 0,C 180,E1 -18422.406,E2 -18422.406} C_VEL
LIN {X 0,Y 268.36,Z 371.277,A -85,B 0,C 180,E1 -18424.086,E2 -18424.086} C_VEL
LIN {X 0,Y 267.249,Z 385.067,A -85,B 0,C 180,E1 -18424.754,E2 -18424.754} C_VEL
LIN {X 0,Y 265.833,Z 398.06,A -85,B 0,C 180,E1 -18425.705,E2 -18425.705} C_VEL
LIN {X 0,Y 264.24,Z 409.886,A -85,B 0,C 180,E1 -18426.902,E2 -18426.902} C_VEL
LIN {X 0,Y 262.424,Z 421.293,A -85,B 0,C 180,E1 -18428.393,E2 -18428.393} C_VEL
LIN {X 0,Y 260.518,Z 431.571,A -85,B 0,C 180,E1 -18430.088,E2 -18430.088} C_VEL
LIN {X 0,Y 258.995,Z 441.148,A -85,B 0,C 180,E1 -18432.099,E2 -18432.099} C_VEL
LIN {X 0,Y 257.432,Z 449.141,A -85,B 0,C 180,E1 -18434.157,E2 -18434.157} C_VEL
LIN {X 0,Y 256.014,Z 456.487,A -85,B 0,C 180,E1 -18436.507,E2 -18436.507} C_VEL
LIN {X 0,Y 255.064,Z 462.365,A -85,B 0,C 180,E1 -18438.88,E2 -18438.88} C_VEL
LIN {X 0,Y 254.458,Z 466.974,A -85,B 0,C 180,E1 -18441.263,E2 -18441.263} C_VEL
LIN {X 0,Y 254.069,Z 470.462,A -85,B 0,C 180,E1 -18443.648,E2 -18443.648} C_VEL
LIN {X 0,Y 253.974,Z 472.198,A -85,B 0,C 180,E1 -18445.238,E2 -18445.238} C_VEL
LIN {X 0,Y 253.979,Z 473.515,A -85,B 0,C 180,E1 -18446.828,E2 -18446.828} C_VEL
LIN {X 0,Y 254.022,Z 474.431,A -85,B 0,C 180,E1 -18448.415,E2 -18448.415} C_VEL
LIN {X 0,Y 254.054,Z 474.935,A -85,B 0,C 180,E1 -18450,E2 -18450} C_VEL
LIN {X 0,Y 254.013,Z 474.999,A -85,B 0,C 180,E1 -18451.586,E2 -18451.586} C_VEL
LIN {X 0,Y 253.974,Z 473.958,A -85,B 0,C 180,E1 -18454.762,E2 -18454.762} C_VEL
LIN {X 0,Y 254.065,Z 472.846,A -85,B 0,C 180,E1 -18456.353,E2 -18456.353} C_VEL
LIN {X 0,Y 254.317,Z 471.284,A -85,B 0,C 180,E1 -18457.942,E2 -18457.942} C_VEL
LIN {X 0,Y 254.922,Z 468.162,A -85,B 0,C 180,E1 -18460.323,E2 -18460.323} C_VEL
LIN {X 0,Y 255.83,Z 463.99,A -85,B 0,C 180,E1 -18462.696,E2 -18462.696} C_VEL
LIN {X 0,Y 257.514,Z 457.641,A -85,B 0,C 180,E1 -18465.432,E2 -18465.432} C_VEL
LIN {X 0,Y 259.361,Z 450.75,A -85,B 0,C 180,E1 -18467.749,E2 -18467.749} C_VEL
LIN {X 0,Y 261.488,Z 442.051,A -85,B 0,C 180,E1 -18470.076,E2 -18470.076} C_VEL
LIN {X 0,Y 263.601,Z 433.43,A -85,B 0,C 180,E1 -18471.917,E2 -18471.917} C_VEL
LIN {X 0,Y 266.159,Z 422.672,A -85,B 0,C 180,E1 -18473.746,E2 -18473.746} C_VEL
LIN {X 0,Y 268.353,Z 411.952,A -85,B 0,C 180,E1 -18475.187,E2 -18475.187} C_VEL
LIN {X 0,Y 270.474,Z 399.976,A -85,B 0,C 180,E1 -18476.422,E2 -18476.422} C_VEL
LIN {X 0,Y 272.189,Z 387.578,A -85,B 0,C 180,E1 -18477.382,E2 -18477.382} C_VEL
LIN {X 0,Y 273.563,Z 374.838,A -85,B 0,C 180,E1 -18478.058,E2 -18478.058} C_VEL
LIN {X 0,Y 274.464,Z 358.816,A -85,B 0,C 180,E1 -18478.566,E2 -18478.566} C_VEL
LIN {X 0,Y 276.098,Z 311.032,A -85,B 0,C 180,E1 -18479.882,E2 -18479.882} C_VEL
LIN {X 0,Y 272.88,Z 290.322,A -85,B 0,C 180,E1 -18481.02,E2 -18481.02} C_VEL
LIN {X 0,Y 272.036,Z 287.247,A -85,B 0,C 180,E1 -18481.248,E2 -18481.248} C_VEL
LIN {X 0,Y 266.079,Z 273.898,A -85,B 0,C 180,E1 -18482.63,E2 -18482.63} C_VEL
LIN {X 0,Y 261.132,Z 264.266,A -85,B 0,C 180,E1 -18483.802,E2 -18483.802} C_VEL
LIN {X 0,Y 259.742,Z 261.213,A -85,B 0,C 180,E1 -18484.196,E2 -18484.196} C_VEL
LIN {X 0,Y 257.673,Z 253.09,A -85,B 0,C 180,E1 -18487.723,E2 -18487.723} C_VEL
LIN {X 0,Y 256.06,Z 247.586,A -85,B 0,C 180,E1 -18490.327,E2 -18490.327} C_VEL
LIN {X 0,Y 256.054,Z 247.589,A -85,B 0,C 180,E1 -18494.469,E2 -18494.469} C_VEL
LIN {X 0,Y 256.055,Z 247.586,A -85,B 0,C 180,E1 -18498.797,E2 -18498.797} C_VEL
LIN {X 0,Y 256.131,Z 247.58,A -85,B 0,C 180,E1 -18502.867,E2 -18502.867} C_VEL
LIN {X 0,Y 256.068,Z 247.588,A -85,B 0,C 180,E1 -18506.707,E2 -18506.707} C_VEL
LIN {X 0,Y 256.114,Z 247.581,A -85,B 0,C 180,E1 -18510.4,E2 -18510.4} C_VEL
LIN {X 0,Y 256.189,Z 247.574,A -85,B 0,C 180,E1 -18514.861,E2 -18514.861} C_VEL
LIN {X 0,Y 256.167,Z 247.578,A -85,B 0,C 180,E1 -18519.105,E2 -18519.105} C_VEL
LIN {X 0,Y 256.3,Z 247.558,A -85,B 0,C 180,E1 -18524.085,E2 -18524.085} C_VEL
LIN {X 0,Y 256.31,Z 247.554,A -85,B 0,C 180,E1 -18528.934,E2 -18528.934} C_VEL
LIN {X 0,Y 256.538,Z 247.526,A -85,B 0,C 180,E1 -18532.127,E2 -18532.127} C_VEL
LIN {X 0,Y 256.714,Z 247.503,A -85,B 0,C 180,E1 -18538.431,E2 -18538.431} C_VEL
LIN {X 0,Y 256.714,Z 247.508,A -85,B 0,C 180,E1 -18541.569,E2 -18541.569} C_VEL
LIN {X 0,Y 256.54,Z 247.52,A -85,B 0,C 180,E1 -18547.873,E2 -18547.873} C_VEL
LIN {X 0,Y 256.31,Z 247.552,A -85,B 0,C 180,E1 -18551.066,E2 -18551.066} C_VEL
LIN {X 0,Y 256.3,Z 247.554,A -85,B 0,C 180,E1 -18555.915,E2 -18555.915} C_VEL
LIN {X 0,Y 256.163,Z 247.573,A -85,B 0,C 180,E1 -18560.896,E2 -18560.896} C_VEL
LIN {X 0,Y 256.16,Z 247.579,A -85,B 0,C 180,E1 -18565.125,E2 -18565.125} C_VEL
LIN {X 0,Y 256.111,Z 247.679,A -85,B 0,C 180,E1 -18568.939,E2 -18568.939} C_VEL
LIN {X 0,Y 256.968,Z 250.801,A -85,B 0,C 180,E1 -18570.396,E2 -18570.396} C_VEL
LIN {X 0,Y 264.666,Z 264.335,A -85,B 0,C 180,E1 -18572.248,E2 -18572.248} C_VEL
LIN {X 0,Y 271.506,Z 278.07,A -85,B 0,C 180,E1 -18573.806,E2 -18573.806} C_VEL
LIN {X 0,Y 276.868,Z 290.856,A -85,B 0,C 180,E1 -18575.015,E2 -18575.015} C_VEL
LIN {X 0,Y 274.134,Z 358.407,A -85,B 0,C 180,E1 -18576.872,E2 -18576.872} C_VEL
LIN {X 0,Y 273.027,Z 371.387,A -85,B 0,C 180,E1 -18577.497,E2 -18577.497} C_VEL
LIN {X 0,Y 271.529,Z 384.045,A -85,B 0,C 180,E1 -18578.404,E2 -18578.404} C_VEL
LIN {X 0,Y 269.861,Z 395.317,A -85,B 0,C 180,E1 -18579.509,E2 -18579.509} C_VEL
LIN {X 0,Y 267.636,Z 407.288,A -85,B 0,C 180,E1 -18581.033,E2 -18581.033} C_VEL
LIN {X 0,Y 265.406,Z 417.523,A -85,B 0,C 180,E1 -18582.685,E2 -18582.685} C_VEL
LIN {X 0,Y 263.309,Z 426.245,A -85,B 0,C 180,E1 -18584.44,E2 -18584.44} C_VEL
LIN {X 0,Y 261.012,Z 434.981,A -85,B 0,C 180,E1 -18586.636,E2 -18586.636} C_VEL
LIN {X 0,Y 259.114,Z 442.07,A -85,B 0,C 180,E1 -18588.873,E2 -18588.873} C_VEL
LIN {X 0,Y 257.527,Z 447.77,A -85,B 0,C 180,E1 -18591.121,E2 -18591.121} C_VEL
LIN {X 0,Y 256.078,Z 453.101,A -85,B 0,C 180,E1 -18593.839,E2 -18593.839} C_VEL
LIN {X 0,Y 255.037,Z 456.921,A -85,B 0,C 180,E1 -18596.555,E2 -18596.555} C_VEL
LIN {X 0,Y 254.36,Z 459.218,A -85,B 0,C 180,E1 -18598.93,E2 -18598.93} C_VEL
LIN {X 0,Y 253.845,Z 460.769,A -85,B 0,C 180,E1 -18601.922,E2 -18601.922} C_VEL
LIN {X 0,Y 253.694,Z 461.048,A -85,B 0,C 180,E1 -18603.689,E2 -18603.689} C_VEL
LIN {X 0,Y 253.653,Z 460.595,A -85,B 0,C 180,E1 -18606.112,E2 -18606.112} C_VEL
LIN {X 0,Y 253.853,Z 458.94,A -85,B 0,C 180,E1 -18608.905,E2 -18608.905} C_VEL
LIN {X 0,Y 254.375,Z 456.256,A -85,B 0,C 180,E1 -18611.474,E2 -18611.474} C_VEL
LIN {X 0,Y 254.975,Z 452.464,A -85,B 0,C 180,E1 -18614,E2 -18614} C_VEL
LIN {X 0,Y 255.819,Z 447.459,A -85,B 0,C 180,E1 -18616.496,E2 -18616.496} C_VEL
LIN {X 0,Y 257.006,Z 441.088,A -85,B 0,C 180,E1 -18618.964,E2 -18618.964} C_VEL
LIN {X 0,Y 258.588,Z 433.108,A -85,B 0,C 180,E1 -18621.403,E2 -18621.403} C_VEL
LIN {X 0,Y 260.184,Z 424.859,A -85,B 0,C 180,E1 -18623.408,E2 -18623.408} C_VEL
LIN {X 0,Y 261.947,Z 414.784,A -85,B 0,C 180,E1 -18625.383,E2 -18625.383} C_VEL
LIN {X 0,Y 263.649,Z 404.822,A -85,B 0,C 180,E1 -18626.944,E2 -18626.944} C_VEL
LIN {X 0,Y 265.172,Z 394.127,A -85,B 0,C 180,E1 -18628.291,E2 -18628.291} C_VEL
LIN {X 0,Y 266.676,Z 381.637,A -85,B 0,C 180,E1 -18629.49,E2 -18629.49} C_VEL
LIN {X 0,Y 267.826,Z 368.335,A -85,B 0,C 180,E1 -18630.423,E2 -18630.423} C_VEL
LIN {X 0,Y 268.602,Z 356.052,A -85,B 0,C 180,E1 -18630.984,E2 -18630.984} C_VEL
LIN {X 0,Y 270.896,Z 286.556,A -85,B 0,C 180,E1 -18632.877,E2 -18632.877} C_VEL
LIN {X 0,Y 269.705,Z 281.963,A -85,B 0,C 180,E1 -18633.133,E2 -18633.133} C_VEL
LIN {X 0,Y 263.048,Z 264.136,A -85,B 0,C 180,E1 -18634.366,E2 -18634.366} C_VEL
LIN {X 0,Y 256.896,Z 249.949,A -85,B 0,C 180,E1 -18635.524,E2 -18635.524} C_VEL
LIN {X 0,Y 256.455,Z 247.543,A -85,B 0,C 180,E1 -18636.589,E2 -18636.589} C_VEL
LIN {X 0,Y 256.429,Z 247.542,A -85,B 0,C 180,E1 -18639.465,E2 -18639.465} C_VEL
LIN {X 0,Y 256.258,Z 247.568,A -85,B 0,C 180,E1 -18644.29,E2 -18644.29} C_VEL
LIN {X 0,Y 256.213,Z 247.575,A -85,B 0,C 180,E1 -18647.561,E2 -18647.561} C_VEL
LIN {X 0,Y 256.155,Z 247.577,A -85,B 0,C 180,E1 -18651.117,E2 -18651.117} C_VEL
LIN {X 0,Y 256.162,Z 247.574,A -85,B 0,C 180,E1 -18655.125,E2 -18655.125} C_VEL
LIN {X 0,Y 256.057,Z 247.584,A -85,B 0,C 180,E1 -18659.606,E2 -18659.606} C_VEL
LIN {X 0,Y 256.066,Z 247.587,A -85,B 0,C 180,E1 -18663.292,E2 -18663.292} C_VEL
LIN {X 0,Y 256.116,Z 247.577,A -85,B 0,C 180,E1 -18667.271,E2 -18667.271} C_VEL
LIN {X 0,Y 256.054,Z 247.587,A -85,B 0,C 180,E1 -18671.203,E2 -18671.203} C_VEL
LIN {X 0,Y 256.054,Z 247.58,A -85,B 0,C 180,E1 -18675.53,E2 -18675.53} C_VEL
LIN {X 0,Y 256.054,Z 247.588,A -85,B 0,C 180,E1 -18678.796,E2 -18678.796} C_VEL
LIN {X 0,Y 256.131,Z 247.569,A -85,B 0,C 180,E1 -18682.867,E2 -18682.867} C_VEL
LIN {X 0,Y 256.067,Z 247.581,A -85,B 0,C 180,E1 -18686.707,E2 -18686.707} C_VEL
LIN {X 0,Y 256.102,Z 247.582,A -85,B 0,C 180,E1 -18690.399,E2 -18690.399} C_VEL
LIN {X 0,Y 256.187,Z 247.557,A -85,B 0,C 180,E1 -18694.861,E2 -18694.861} C_VEL
LIN {X 0,Y 256.165,Z 247.567,A -85,B 0,C 180,E1 -18699.105,E2 -18699.105} C_VEL
LIN {X 0,Y 256.298,Z 247.558,A -85,B 0,C 180,E1 -18704.085,E2 -18704.085} C_VEL
LIN {X 0,Y 256.308,Z 247.535,A -85,B 0,C 180,E1 -18708.934,E2 -18708.934} C_VEL
LIN {X 0,Y 256.538,Z 247.522,A -85,B 0,C 180,E1 -18712.127,E2 -18712.127} C_VEL
LIN {X 0,Y 256.713,Z 247.502,A -85,B 0,C 180,E1 -18718.431,E2 -18718.431} C_VEL
LIN {X 0,Y 256.712,Z 247.491,A -85,B 0,C 180,E1 -18721.569,E2 -18721.569} C_VEL
LIN {X 0,Y 256.388,Z 247.542,A -85,B 0,C 180,E1 -18725.511,E2 -18725.511} C_VEL
LIN {X 0,Y 255.793,Z 247.622,A -85,B 0,C 180,E1 -18726.823,E2 -18726.823} C_VEL
LIN {X 0,Y 254.203,Z 247.822,A -85,B 0,C 180,E1 -18728.11,E2 -18728.11} C_VEL
LIN {X 0,Y 250.371,Z 248.291,A -85,B 0,C 180,E1 -18730.699,E2 -18730.699} C_VEL
LIN {X 0,Y 249.291,Z 248.421,A -85,B 0,C 180,E1 -18732.051,E2 -18732.051} C_VEL
LIN {X 0,Y 249.207,Z 248.425,A -85,B 0,C 180,E1 -18732.51,E2 -18732.51} C_VEL
LIN {X 0,Y 249.216,Z 248.439,A -85,B 0,C 180,E1 -18736.503,E2 -18736.503} C_VEL
LIN {X 0,Y 249.085,Z 248.452,A -85,B 0,C 180,E1 -18741.518,E2 -18741.518} C_VEL
LIN {X 0,Y 249.129,Z 248.451,A -85,B 0,C 180,E1 -18745.482,E2 -18745.482} C_VEL
LIN {X 0,Y 249.082,Z 248.454,A -85,B 0,C 180,E1 -18748.994,E2 -18748.994} C_VEL
LIN {X 0,Y 249.029,Z 248.464,A -85,B 0,C 180,E1 -18752.426,E2 -18752.426} C_VEL
LIN {X 0,Y 249.047,Z 248.464,A -85,B 0,C 180,E1 -18756.343,E2 -18756.343} C_VEL
LIN {X 0,Y 249.004,Z 248.467,A -85,B 0,C 180,E1 -18760.478,E2 -18760.478} C_VEL
LIN {X 0,Y 248.993,Z 248.471,A -85,B 0,C 180,E1 -18764.882,E2 -18764.882} C_VEL
LIN {X 0,Y 249.018,Z 248.466,A -85,B 0,C 180,E1 -18767.364,E2 -18767.364} C_VEL
LIN {X 0,Y 249.039,Z 248.459,A -85,B 0,C 180,E1 -18771.622,E2 -18771.622} C_VEL
LIN {X 0,Y 249.129,Z 248.579,A -85,B 0,C 180,E1 -18773.421,E2 -18773.421} C_VEL
LIN {X 0,Y 251.317,Z 258.404,A -85,B 0,C 180,E1 -18777.374,E2 -18777.374} C_VEL
LIN {X 0,Y 252.213,Z 262.639,A -85,B 0,C 180,E1 -18779.002,E2 -18779.002} C_VEL
LIN {X 0,Y 259.485,Z 281.679,A -85,B 0,C 180,E1 -18780.427,E2 -18780.427} C_VEL
LIN {X 0,Y 263.753,Z 310.134,A -85,B 0,C 180,E1 -18781.762,E2 -18781.762} C_VEL
LIN {X 0,Y 262.569,Z 350.865,A -85,B 0,C 180,E1 -18782.902,E2 -18782.902} C_VEL
LIN {X 0,Y 261.659,Z 373.351,A -85,B 0,C 180,E1 -18783.586,E2 -18783.586} C_VEL
LIN {X 0,Y 260.623,Z 385.656,A -85,B 0,C 180,E1 -18784.226,E2 -18784.226} C_VEL
LIN {X 0,Y 259.226,Z 397.882,A -85,B 0,C 180,E1 -18785.151,E2 -18785.151} C_VEL
LIN {X 0,Y 257.436,Z 410.495,A -85,B 0,C 180,E1 -18786.468,E2 -18786.468} C_VEL
LIN {X 0,Y 255.576,Z 421.758,A -85,B 0,C 180,E1 -18787.997,E2 -18787.997} C_VEL
LIN {X 0,Y 253.612,Z 431.879,A -85,B 0,C 180,E1 -18789.733,E2 -18789.733} C_VEL
LIN {X 0,Y 252.031,Z 441.431,A -85,B 0,C 180,E1 -18791.812,E2 -18791.812} C_VEL
LIN {X 0,Y 250.323,Z 449.982,A -85,B 0,C 180,E1 -18794.114,E2 -18794.114} C_VEL
LIN {X 0,Y 248.868,Z 457.112,A -85,B 0,C 180,E1 -18796.528,E2 -18796.528} C_VEL
LIN {X 0,Y 247.798,Z 463.614,A -85,B 0,C 180,E1 -18799.377,E2 -18799.377} C_VEL
LIN {X 0,Y 247.258,Z 467.886,A -85,B 0,C 180,E1 -18801.83,E2 -18801.83} C_VEL
LIN {X 0,Y 247.011,Z 470.143,A -85,B 0,C 180,E1 -18803.465,E2 -18803.465} C_VEL
LIN {X 0,Y 246.902,Z 471.914,A -85,B 0,C 180,E1 -18805.102,E2 -18805.102} C_VEL
LIN {X 0,Y 246.879,Z 473.251,A -85,B 0,C 180,E1 -18806.736,E2 -18806.736} C_VEL
LIN {X 0,Y 246.93,Z 474.186,A -85,B 0,C 180,E1 -18808.369,E2 -18808.369} C_VEL
LIN {X 0,Y 246.983,Z 474.721,A -85,B 0,C 180,E1 -18810,E2 -18810} C_VEL
LIN {X 0,Y 246.921,Z 474.811,A -85,B 0,C 180,E1 -18811.631,E2 -18811.631} C_VEL
LIN {X 0,Y 246.883,Z 473.807,A -85,B 0,C 180,E1 -18814.899,E2 -18814.899} C_VEL
LIN {X 0,Y 247.01,Z 472.721,A -85,B 0,C 180,E1 -18816.535,E2 -18816.535} C_VEL
LIN {X 0,Y 247.268,Z 471.189,A -85,B 0,C 180,E1 -18818.17,E2 -18818.17} C_VEL
LIN {X 0,Y 247.901,Z 468.106,A -85,B 0,C 180,E1 -18820.619,E2 -18820.619} C_VEL
LIN {X 0,Y 248.872,Z 463.984,A -85,B 0,C 180,E1 -18823.057,E2 -18823.057} C_VEL
LIN {X 0,Y 250.66,Z 457.694,A -85,B 0,C 180,E1 -18825.865,E2 -18825.865} C_VEL
LIN {X 0,Y 252.567,Z 450.873,A -85,B 0,C 180,E1 -18828.243,E2 -18828.243} C_VEL
LIN {X 0,Y 254.795,Z 442.411,A -85,B 0,C 180,E1 -18830.592,E2 -18830.592} C_VEL
LIN {X 0,Y 257.029,Z 433.738,A -85,B 0,C 180,E1 -18832.508,E2 -18832.508} C_VEL
LIN {X 0,Y 259.701,Z 423.079,A -85,B 0,C 180,E1 -18834.374,E2 -18834.374} C_VEL
LIN {X 0,Y 261.988,Z 412.523,A -85,B 0,C 180,E1 -18835.844,E2 -18835.844} C_VEL
LIN {X 0,Y 264.179,Z 400.796,A -85,B 0,C 180,E1 -18837.102,E2 -18837.102} C_VEL
LIN {X 0,Y 266.118,Z 387.43,A -85,B 0,C 180,E1 -18838.169,E2 -18838.169} C_VEL
LIN {X 0,Y 267.555,Z 374.378,A -85,B 0,C 180,E1 -18838.871,E2 -18838.871} C_VEL
LIN {X 0,Y 268.51,Z 357.401,A -85,B 0,C 180,E1 -18839.413,E2 -18839.413} C_VEL
LIN {X 0,Y 270.197,Z 312.063,A -85,B 0,C 180,E1 -18840.686,E2 -18840.686} C_VEL
LIN {X 0,Y 267.307,Z 292.934,A -85,B 0,C 180,E1 -18841.775,E2 -18841.775} C_VEL
LIN {X 0,Y 266.321,Z 289.584,A -85,B 0,C 180,E1 -18842.046,E2 -18842.046} C_VEL
LIN {X 0,Y 259.21,Z 273.984,A -85,B 0,C 180,E1 -18843.779,E2 -18843.779} C_VEL
LIN {X 0,Y 254.202,Z 264.528,A -85,B 0,C 180,E1 -18845.042,E2 -18845.042} C_VEL
LIN {X 0,Y 252.458,Z 260.935,A -85,B 0,C 180,E1 -18845.554,E2 -18845.554} C_VEL
LIN {X 0,Y 250.882,Z 254.83,A -85,B 0,C 180,E1 -18848.338,E2 -18848.338} C_VEL
LIN {X 0,Y 249.019,Z 248.467,A -85,B 0,C 180,E1 -18851.546,E2 -18851.546} C_VEL
LIN {X 0,Y 248.993,Z 248.466,A -85,B 0,C 180,E1 -18855.119,E2 -18855.119} C_VEL
LIN {X 0,Y 249.016,Z 248.464,A -85,B 0,C 180,E1 -18857.363,E2 -18857.363} C_VEL
LIN {X 0,Y 249.044,Z 248.459,A -85,B 0,C 180,E1 -18862.2,E2 -18862.2} C_VEL
LIN {X 0,Y 249.044,Z 248.456,A -85,B 0,C 180,E1 -18865.639,E2 -18865.639} C_VEL
LIN {X 0,Y 249.052,Z 248.454,A -85,B 0,C 180,E1 -18869.473,E2 -18869.473} C_VEL
LIN {X 0,Y 249.074,Z 248.449,A -85,B 0,C 180,E1 -18873.162,E2 -18873.162} C_VEL
LIN {X 0,Y 249.08,Z 248.448,A -85,B 0,C 180,E1 -18876.733,E2 -18876.733} C_VEL
LIN {X 0,Y 249.111,Z 248.45,A -85,B 0,C 180,E1 -18880.212,E2 -18880.212} C_VEL
LIN {X 0,Y 249.242,Z 248.438,A -85,B 0,C 180,E1 -18883.622,E2 -18883.622} C_VEL
LIN {X 0,Y 249.253,Z 248.437,A -85,B 0,C 180,E1 -18888.617,E2 -18888.617} C_VEL
LIN {X 0,Y 249.48,Z 248.405,A -85,B 0,C 180,E1 -18891.903,E2 -18891.903} C_VEL
LIN {X 0,Y 249.436,Z 248.412,A -85,B 0,C 180,E1 -18896.77,E2 -18896.77} C_VEL
LIN {X 0,Y 249.722,Z 248.367,A -85,B 0,C 180,E1 -18900,E2 -18900} C_VEL
LIN {X 0,Y 249.435,Z 248.406,A -85,B 0,C 180,E1 -18903.231,E2 -18903.231} C_VEL
LIN {X 0,Y 249.482,Z 248.399,A -85,B 0,C 180,E1 -18908.097,E2 -18908.097} C_VEL
LIN {X 0,Y 249.253,Z 248.429,A -85,B 0,C 180,E1 -18911.384,E2 -18911.384} C_VEL
LIN {X 0,Y 249.243,Z 248.437,A -85,B 0,C 180,E1 -18916.378,E2 -18916.378} C_VEL
LIN {X 0,Y 249.084,Z 248.455,A -85,B 0,C 180,E1 -18921.519,E2 -18921.519} C_VEL
LIN {X 0,Y 249.105,Z 248.456,A -85,B 0,C 180,E1 -18925.469,E2 -18925.469} C_VEL
LIN {X 0,Y 249.065,Z 248.534,A -85,B 0,C 180,E1 -18927.749,E2 -18927.749} C_VEL
LIN {X 0,Y 249.742,Z 251.026,A -85,B 0,C 180,E1 -18929.003,E2 -18929.003} C_VEL
LIN {X 0,Y 252.142,Z 255.062,A -85,B 0,C 180,E1 -18929.641,E2 -18929.641} C_VEL
LIN {X 0,Y 259.347,Z 267.545,A -85,B 0,C 180,E1 -18931.452,E2 -18931.452} C_VEL
